// TwinCAT 3 PLC project PLC1
// ProgramVersion: 3.1.4026.16
// libraries:
//   SPT Base Types, * (Beckhoff Automation LLC)
//   Tc2_Standard, * (Beckhoff Automation GmbH)
//   Tc2_System, * (Beckhoff Automation GmbH)
//   Tc3_Module, * (Beckhoff Automation GmbH)
//   Tc3_PackML_V2, * (Beckhoff Automation GmbH)
//   Tc3_XPlanarUtility, * (Beckhoff Automation GmbH)
//   XPlanarApplication, * (Beckhoff Automation LLC)
// project tree:
//   / GlobalTextList.TcGTLO (not stored), PlcTask.TcTTO, Visualization Manager.TcVMO (not stored)
//   POUs/CustomStations/ FB_BounceStation.TcPOU, FB_RotateStation.TcPOU (not stored), FB_TiltStation.TcPOU
//   POUs/ FB_XPlanarModule.TcPOU, MAIN.TcPOU
//   POUs/Utilities/ ErrorStep.TcPOU (not stored), NextMinorStep.TcPOU (not stored), NextStep.TcPOU (not stored)
//   VISUs/ V_Main.TcVIS
// real-time tasks:
//   TASK MC-Task (MET): cycle T#2ms, priority 6, ADS port 355
//   TASK MC-Task (MPT): cycle T#10ms, priority 7, ADS port 356
//   TASK Job Task: cycle default, priority 8
//   TASK PlcTask: cycle T#10ms, priority 20, ADS port 352
//   TASK XPlanar Task_3: cycle T#250us, priority 1, ADS port 350
//   TASK XPlanar Task_4: cycle T#250us, priority 2, ADS port 351
// I/O:
//   DEVICE Device 1 (EtherCAT), AmsNetId 5.85.147.112.2.1
//     Term 1 (EK1200) [EK1200-5000 EtherCAT Power supply (2A E-Bus)]
//       Term 2 (EL9222-9482) [EL9222-9482 Overcurrent protection 24V DC, 2Ch., 8A/2A]
//       Term 3 (EL9222-6600) [EL9222-6600 Overcurrent protection 24V DC, 2Ch., max. 4A, adjustable]
//       Term 4 (EL9011) [EL9011 End Terminal]
//   DEVICE Device 4 (EtherCAT), AmsNetId 5.85.147.112.5.1
//     Term 5 (APS4322-7000) [APS4322-7000 Drive]
//       Term 6 (APS4322-5000) [APS4322-5000 Feedback]
//     Term 7 (APS4322-7000) [APS4322-7000 Drive]
//       Term 8 (APS4322-5000) [APS4322-5000 Feedback]
//     Term 9 (APS4322-7000) [APS4322-7000 Drive]
//       Term 10 (APS4322-5000) [APS4322-5000 Feedback]
//     Term 11 (APS4322-7000) [APS4322-7000 Drive]
//       Term 12 (APS4322-5000) [APS4322-5000 Feedback]
//     Term 13 (APS4322-7000) [APS4322-7000 Drive]
//       Term 14 (APS4322-5000) [APS4322-5000 Feedback]
//     Term 15 (APS4322-7000) [APS4322-7000 Drive]
//       Term 16 (APS4322-5000) [APS4322-5000 Feedback]
// variable links:
//   Device 4 (EtherCAT) <-> TcCOM Objects/XPlanar/Part1/Tile1
//     Term 5 (APS4322-7000)/APS Comm Inputs/CommStatusWord <-> Data Pointer/MoverCommStatusWord
//     Term 5 (APS4322-7000)/APS Comm Inputs/Data {1..4} <-> Data Pointer/MoverCommDataIn[{0..3}]  (4 links)
//     Term 5 (APS4322-7000)/APS Comm Outputs/CommControlWord <-> Data Pointer/MoverCommControlWord
//     Term 5 (APS4322-7000)/APS Comm Outputs/Data 1 <-> Data Pointer/MoverCommDataOut
//     Term 5 (APS4322-7000)/APS Diagdata/DC Link Voltage <-> Data Pointer/DcLinkVoltage
//     Term 5 (APS4322-7000)/APS Diagdata/Power supply current <-> Data Pointer/PowerSupplyCurrent
//     Term 5 (APS4322-7000)/APS Inputs/StatusWord <-> Data Pointer/PowerUnitStatusWord
//     Term 5 (APS4322-7000)/APS Outputs/ControlWord <-> Data Pointer/PowerUnitControlWord
//     Term 5 (APS4322-7000)/APS Outputs/Current D 0X0 <-> Data Pointer/DCurrentSetPoints[0]
//     Term 5 (APS4322-7000)/APS Outputs/Current D 0X1 <-> Data Pointer/DCurrentSetPoints[1]
//     Term 5 (APS4322-7000)/APS Outputs/Current D 0X2 <-> Data Pointer/DCurrentSetPoints[2]
//     Term 5 (APS4322-7000)/APS Outputs/Current D 1X0 <-> Data Pointer/DCurrentSetPoints[6]
//     Term 5 (APS4322-7000)/APS Outputs/Current D 1X1 <-> Data Pointer/DCurrentSetPoints[7]
//     Term 5 (APS4322-7000)/APS Outputs/Current D 1X2 <-> Data Pointer/DCurrentSetPoints[8]
//     Term 5 (APS4322-7000)/APS Outputs/Current D 2X0 <-> Data Pointer/DCurrentSetPoints[12]
//     Term 5 (APS4322-7000)/APS Outputs/Current D 2X1 <-> Data Pointer/DCurrentSetPoints[13]
//     Term 5 (APS4322-7000)/APS Outputs/Current D 2X2 <-> Data Pointer/DCurrentSetPoints[14]
//     Term 5 (APS4322-7000)/APS Outputs/Current D 3X0 <-> Data Pointer/DCurrentSetPoints[18]
//     Term 5 (APS4322-7000)/APS Outputs/Current D 3X1 <-> Data Pointer/DCurrentSetPoints[19]
//     Term 5 (APS4322-7000)/APS Outputs/Current D 3X2 <-> Data Pointer/DCurrentSetPoints[20]
//     Term 5 (APS4322-7000)/APS Outputs/Current D 0Y0 <-> Data Pointer/DCurrentSetPoints[3]
//     Term 5 (APS4322-7000)/APS Outputs/Current D 0Y1 <-> Data Pointer/DCurrentSetPoints[4]
//     Term 5 (APS4322-7000)/APS Outputs/Current D 0Y2 <-> Data Pointer/DCurrentSetPoints[5]
//     Term 5 (APS4322-7000)/APS Outputs/Current D 1Y0 <-> Data Pointer/DCurrentSetPoints[9]
//     Term 5 (APS4322-7000)/APS Outputs/Current D 1Y1 <-> Data Pointer/DCurrentSetPoints[10]
//     Term 5 (APS4322-7000)/APS Outputs/Current D 1Y2 <-> Data Pointer/DCurrentSetPoints[11]
//     Term 5 (APS4322-7000)/APS Outputs/Current D 2Y0 <-> Data Pointer/DCurrentSetPoints[15]
//     Term 5 (APS4322-7000)/APS Outputs/Current D 2Y1 <-> Data Pointer/DCurrentSetPoints[16]
//     Term 5 (APS4322-7000)/APS Outputs/Current D 2Y2 <-> Data Pointer/DCurrentSetPoints[17]
//     Term 5 (APS4322-7000)/APS Outputs/Current D 3Y0 <-> Data Pointer/DCurrentSetPoints[21]
//     Term 5 (APS4322-7000)/APS Outputs/Current D 3Y1 <-> Data Pointer/DCurrentSetPoints[22]
//     Term 5 (APS4322-7000)/APS Outputs/Current D 3Y2 <-> Data Pointer/DCurrentSetPoints[23]
//     Term 5 (APS4322-7000)/APS Outputs/Current Q 0X0 <-> Data Pointer/QCurrentSetPoints[0]
//     Term 5 (APS4322-7000)/APS Outputs/Current Q 0X1 <-> Data Pointer/QCurrentSetPoints[1]
//     Term 5 (APS4322-7000)/APS Outputs/Current Q 0X2 <-> Data Pointer/QCurrentSetPoints[2]
//     Term 5 (APS4322-7000)/APS Outputs/Current Q 1X0 <-> Data Pointer/QCurrentSetPoints[6]
//     Term 5 (APS4322-7000)/APS Outputs/Current Q 1X1 <-> Data Pointer/QCurrentSetPoints[7]
//     Term 5 (APS4322-7000)/APS Outputs/Current Q 1X2 <-> Data Pointer/QCurrentSetPoints[8]
//     Term 5 (APS4322-7000)/APS Outputs/Current Q 2X0 <-> Data Pointer/QCurrentSetPoints[12]
//     Term 5 (APS4322-7000)/APS Outputs/Current Q 2X1 <-> Data Pointer/QCurrentSetPoints[13]
//     Term 5 (APS4322-7000)/APS Outputs/Current Q 2X2 <-> Data Pointer/QCurrentSetPoints[14]
//     Term 5 (APS4322-7000)/APS Outputs/Current Q 3X0 <-> Data Pointer/QCurrentSetPoints[18]
//     Term 5 (APS4322-7000)/APS Outputs/Current Q 3X1 <-> Data Pointer/QCurrentSetPoints[19]
//     Term 5 (APS4322-7000)/APS Outputs/Current Q 3X2 <-> Data Pointer/QCurrentSetPoints[20]
//     Term 5 (APS4322-7000)/APS Outputs/Current Q 0Y0 <-> Data Pointer/QCurrentSetPoints[3]
//     Term 5 (APS4322-7000)/APS Outputs/Current Q 0Y1 <-> Data Pointer/QCurrentSetPoints[4]
//     Term 5 (APS4322-7000)/APS Outputs/Current Q 0Y2 <-> Data Pointer/QCurrentSetPoints[5]
//     Term 5 (APS4322-7000)/APS Outputs/Current Q 1Y0 <-> Data Pointer/QCurrentSetPoints[9]
//     Term 5 (APS4322-7000)/APS Outputs/Current Q 1Y1 <-> Data Pointer/QCurrentSetPoints[10]
//     Term 5 (APS4322-7000)/APS Outputs/Current Q 1Y2 <-> Data Pointer/QCurrentSetPoints[11]
//     Term 5 (APS4322-7000)/APS Outputs/Current Q 2Y0 <-> Data Pointer/QCurrentSetPoints[15]
//     Term 5 (APS4322-7000)/APS Outputs/Current Q 2Y1 <-> Data Pointer/QCurrentSetPoints[16]
//     Term 5 (APS4322-7000)/APS Outputs/Current Q 2Y2 <-> Data Pointer/QCurrentSetPoints[17]
//     Term 5 (APS4322-7000)/APS Outputs/Current Q 3Y0 <-> Data Pointer/QCurrentSetPoints[21]
//     Term 5 (APS4322-7000)/APS Outputs/Current Q 3Y1 <-> Data Pointer/QCurrentSetPoints[22]
//     Term 5 (APS4322-7000)/APS Outputs/Current Q 3Y2 <-> Data Pointer/QCurrentSetPoints[23]
//     Term 5 (APS4322-7000)/APS Outputs/PhiE 0X0 <-> Data Pointer/PhiSetPoints[0]
//     Term 5 (APS4322-7000)/APS Outputs/PhiE 0X1 <-> Data Pointer/PhiSetPoints[1]
//     Term 5 (APS4322-7000)/APS Outputs/PhiE 0X2 <-> Data Pointer/PhiSetPoints[2]
//     Term 5 (APS4322-7000)/APS Outputs/PhiE 1X0 <-> Data Pointer/PhiSetPoints[6]
//     Term 5 (APS4322-7000)/APS Outputs/PhiE 1X1 <-> Data Pointer/PhiSetPoints[7]
//     Term 5 (APS4322-7000)/APS Outputs/PhiE 1X2 <-> Data Pointer/PhiSetPoints[8]
//     Term 5 (APS4322-7000)/APS Outputs/PhiE 2X0 <-> Data Pointer/PhiSetPoints[12]
//     Term 5 (APS4322-7000)/APS Outputs/PhiE 2X1 <-> Data Pointer/PhiSetPoints[13]
//     Term 5 (APS4322-7000)/APS Outputs/PhiE 2X2 <-> Data Pointer/PhiSetPoints[14]
//     Term 5 (APS4322-7000)/APS Outputs/PhiE 3X0 <-> Data Pointer/PhiSetPoints[18]
//     Term 5 (APS4322-7000)/APS Outputs/PhiE 3X1 <-> Data Pointer/PhiSetPoints[19]
//     Term 5 (APS4322-7000)/APS Outputs/PhiE 3X2 <-> Data Pointer/PhiSetPoints[20]
//     Term 5 (APS4322-7000)/APS Outputs/PhiE 0Y0 <-> Data Pointer/PhiSetPoints[3]
//     Term 5 (APS4322-7000)/APS Outputs/PhiE 0Y1 <-> Data Pointer/PhiSetPoints[4]
//     Term 5 (APS4322-7000)/APS Outputs/PhiE 0Y2 <-> Data Pointer/PhiSetPoints[5]
//     Term 5 (APS4322-7000)/APS Outputs/PhiE 1Y0 <-> Data Pointer/PhiSetPoints[9]
//     Term 5 (APS4322-7000)/APS Outputs/PhiE 1Y1 <-> Data Pointer/PhiSetPoints[10]
//     Term 5 (APS4322-7000)/APS Outputs/PhiE 1Y2 <-> Data Pointer/PhiSetPoints[11]
//     Term 5 (APS4322-7000)/APS Outputs/PhiE 2Y0 <-> Data Pointer/PhiSetPoints[15]
//     Term 5 (APS4322-7000)/APS Outputs/PhiE 2Y1 <-> Data Pointer/PhiSetPoints[16]
//     Term 5 (APS4322-7000)/APS Outputs/PhiE 2Y2 <-> Data Pointer/PhiSetPoints[17]
//     Term 5 (APS4322-7000)/APS Outputs/PhiE 3Y0 <-> Data Pointer/PhiSetPoints[21]
//     Term 5 (APS4322-7000)/APS Outputs/PhiE 3Y1 <-> Data Pointer/PhiSetPoints[22]
//     Term 5 (APS4322-7000)/APS Outputs/PhiE 3Y2 <-> Data Pointer/PhiSetPoints[23]
//     Term 5 (APS4322-7000)/Term 6 (APS4322-5000)/FB Inputs/A{0..8 step 2} X-Field <-> Data Pointer/HallSensorFieldsXYZ[{0..12 step 3}]  (5 links)
//     Term 5 (APS4322-7000)/Term 6 (APS4322-5000)/FB Inputs/A{0..8 step 2} Y-Field <-> Data Pointer/HallSensorFieldsXYZ[{1..13 step 3}]  (5 links)
//     Term 5 (APS4322-7000)/Term 6 (APS4322-5000)/FB Inputs/A{0..8 step 2} Z-Field <-> Data Pointer/HallSensorFieldsXYZ[{2..14 step 3}]  (5 links)
//     Term 5 (APS4322-7000)/Term 6 (APS4322-5000)/FB Inputs/B{1..9 step 2} X-Field <-> Data Pointer/HallSensorFieldsXYZ[{15..27 step 3}]  (5 links)
//     Term 5 (APS4322-7000)/Term 6 (APS4322-5000)/FB Inputs/B{1..9 step 2} Y-Field <-> Data Pointer/HallSensorFieldsXYZ[{16..28 step 3}]  (5 links)
//     Term 5 (APS4322-7000)/Term 6 (APS4322-5000)/FB Inputs/B{1..9 step 2} Z-Field <-> Data Pointer/HallSensorFieldsXYZ[{17..29 step 3}]  (5 links)
//     Term 5 (APS4322-7000)/Term 6 (APS4322-5000)/FB Inputs/C{0..8 step 2} X-Field <-> Data Pointer/HallSensorFieldsXYZ[{30..42 step 3}]  (5 links)
//     Term 5 (APS4322-7000)/Term 6 (APS4322-5000)/FB Inputs/C{0..8 step 2} Y-Field <-> Data Pointer/HallSensorFieldsXYZ[{31..43 step 3}]  (5 links)
//     Term 5 (APS4322-7000)/Term 6 (APS4322-5000)/FB Inputs/C{0..8 step 2} Z-Field <-> Data Pointer/HallSensorFieldsXYZ[{32..44 step 3}]  (5 links)
//     Term 5 (APS4322-7000)/Term 6 (APS4322-5000)/FB Inputs/D{1..9 step 2} X-Field <-> Data Pointer/HallSensorFieldsXYZ[{45..57 step 3}]  (5 links)
//     Term 5 (APS4322-7000)/Term 6 (APS4322-5000)/FB Inputs/D{1..9 step 2} Y-Field <-> Data Pointer/HallSensorFieldsXYZ[{46..58 step 3}]  (5 links)
//     Term 5 (APS4322-7000)/Term 6 (APS4322-5000)/FB Inputs/D{1..9 step 2} Z-Field <-> Data Pointer/HallSensorFieldsXYZ[{47..59 step 3}]  (5 links)
//     Term 5 (APS4322-7000)/Term 6 (APS4322-5000)/FB Inputs/E{0..8 step 2} X-Field <-> Data Pointer/HallSensorFieldsXYZ[{60..72 step 3}]  (5 links)
//     Term 5 (APS4322-7000)/Term 6 (APS4322-5000)/FB Inputs/E{0..8 step 2} Y-Field <-> Data Pointer/HallSensorFieldsXYZ[{61..73 step 3}]  (5 links)
//     Term 5 (APS4322-7000)/Term 6 (APS4322-5000)/FB Inputs/E{0..8 step 2} Z-Field <-> Data Pointer/HallSensorFieldsXYZ[{62..74 step 3}]  (5 links)
//     Term 5 (APS4322-7000)/Term 6 (APS4322-5000)/FB Inputs/F{1..9 step 2} X-Field <-> Data Pointer/HallSensorFieldsXYZ[{75..87 step 3}]  (5 links)
//     Term 5 (APS4322-7000)/Term 6 (APS4322-5000)/FB Inputs/F{1..9 step 2} Y-Field <-> Data Pointer/HallSensorFieldsXYZ[{76..88 step 3}]  (5 links)
//     Term 5 (APS4322-7000)/Term 6 (APS4322-5000)/FB Inputs/F{1..9 step 2} Z-Field <-> Data Pointer/HallSensorFieldsXYZ[{77..89 step 3}]  (5 links)
//     Term 5 (APS4322-7000)/Term 6 (APS4322-5000)/FB Inputs/G{0..8 step 2} X-Field <-> Data Pointer/HallSensorFieldsXYZ[{90..102 step 3}]  (5 links)
//     Term 5 (APS4322-7000)/Term 6 (APS4322-5000)/FB Inputs/G{0..8 step 2} Y-Field <-> Data Pointer/HallSensorFieldsXYZ[{91..103 step 3}]  (5 links)
//     Term 5 (APS4322-7000)/Term 6 (APS4322-5000)/FB Inputs/G{0..8 step 2} Z-Field <-> Data Pointer/HallSensorFieldsXYZ[{92..104 step 3}]  (5 links)
//     Term 5 (APS4322-7000)/Term 6 (APS4322-5000)/FB Inputs/H{1..9 step 2} X-Field <-> Data Pointer/HallSensorFieldsXYZ[{105..117 step 3}]  (5 links)
//     Term 5 (APS4322-7000)/Term 6 (APS4322-5000)/FB Inputs/H{1..9 step 2} Y-Field <-> Data Pointer/HallSensorFieldsXYZ[{106..118 step 3}]  (5 links)
//     Term 5 (APS4322-7000)/Term 6 (APS4322-5000)/FB Inputs/H{1..9 step 2} Z-Field <-> Data Pointer/HallSensorFieldsXYZ[{107..119 step 3}]  (5 links)
//     Term 5 (APS4322-7000)/Term 6 (APS4322-5000)/FB Inputs/I{0..8 step 2} X-Field <-> Data Pointer/HallSensorFieldsXYZ[{120..132 step 3}]  (5 links)
//     Term 5 (APS4322-7000)/Term 6 (APS4322-5000)/FB Inputs/I{0..8 step 2} Y-Field <-> Data Pointer/HallSensorFieldsXYZ[{121..133 step 3}]  (5 links)
//     Term 5 (APS4322-7000)/Term 6 (APS4322-5000)/FB Inputs/I{0..8 step 2} Z-Field <-> Data Pointer/HallSensorFieldsXYZ[{122..134 step 3}]  (5 links)
//     Term 5 (APS4322-7000)/Term 6 (APS4322-5000)/FB Inputs/J{1..9 step 2} X-Field <-> Data Pointer/HallSensorFieldsXYZ[{135..147 step 3}]  (5 links)
//     Term 5 (APS4322-7000)/Term 6 (APS4322-5000)/FB Inputs/J{1..9 step 2} Y-Field <-> Data Pointer/HallSensorFieldsXYZ[{136..148 step 3}]  (5 links)
//     Term 5 (APS4322-7000)/Term 6 (APS4322-5000)/FB Inputs/J{1..9 step 2} Z-Field <-> Data Pointer/HallSensorFieldsXYZ[{137..149 step 3}]  (5 links)
//     Term 5 (APS4322-7000)/Term 6 (APS4322-5000)/FB Inputs/Status <-> Data Pointer/FeedbackStatus
//   Device 4 (EtherCAT) <-> TcCOM Objects/XPlanar/Part1/Tile2
//     Term 7 (APS4322-7000)/APS Comm Inputs/CommStatusWord <-> Data Pointer/MoverCommStatusWord
//     Term 7 (APS4322-7000)/APS Comm Inputs/Data {1..4} <-> Data Pointer/MoverCommDataIn[{0..3}]  (4 links)
//     Term 7 (APS4322-7000)/APS Comm Outputs/CommControlWord <-> Data Pointer/MoverCommControlWord
//     Term 7 (APS4322-7000)/APS Comm Outputs/Data 1 <-> Data Pointer/MoverCommDataOut
//     Term 7 (APS4322-7000)/APS Diagdata/DC Link Voltage <-> Data Pointer/DcLinkVoltage
//     Term 7 (APS4322-7000)/APS Diagdata/Power supply current <-> Data Pointer/PowerSupplyCurrent
//     Term 7 (APS4322-7000)/APS Inputs/StatusWord <-> Data Pointer/PowerUnitStatusWord
//     Term 7 (APS4322-7000)/APS Outputs/ControlWord <-> Data Pointer/PowerUnitControlWord
//     Term 7 (APS4322-7000)/APS Outputs/Current D 0X0 <-> Data Pointer/DCurrentSetPoints[0]
//     Term 7 (APS4322-7000)/APS Outputs/Current D 0X1 <-> Data Pointer/DCurrentSetPoints[1]
//     Term 7 (APS4322-7000)/APS Outputs/Current D 0X2 <-> Data Pointer/DCurrentSetPoints[2]
//     Term 7 (APS4322-7000)/APS Outputs/Current D 1X0 <-> Data Pointer/DCurrentSetPoints[6]
//     Term 7 (APS4322-7000)/APS Outputs/Current D 1X1 <-> Data Pointer/DCurrentSetPoints[7]
//     Term 7 (APS4322-7000)/APS Outputs/Current D 1X2 <-> Data Pointer/DCurrentSetPoints[8]
//     Term 7 (APS4322-7000)/APS Outputs/Current D 2X0 <-> Data Pointer/DCurrentSetPoints[12]
//     Term 7 (APS4322-7000)/APS Outputs/Current D 2X1 <-> Data Pointer/DCurrentSetPoints[13]
//     Term 7 (APS4322-7000)/APS Outputs/Current D 2X2 <-> Data Pointer/DCurrentSetPoints[14]
//     Term 7 (APS4322-7000)/APS Outputs/Current D 3X0 <-> Data Pointer/DCurrentSetPoints[18]
//     Term 7 (APS4322-7000)/APS Outputs/Current D 3X1 <-> Data Pointer/DCurrentSetPoints[19]
//     Term 7 (APS4322-7000)/APS Outputs/Current D 3X2 <-> Data Pointer/DCurrentSetPoints[20]
//     Term 7 (APS4322-7000)/APS Outputs/Current D 0Y0 <-> Data Pointer/DCurrentSetPoints[3]
//     Term 7 (APS4322-7000)/APS Outputs/Current D 0Y1 <-> Data Pointer/DCurrentSetPoints[4]
//     Term 7 (APS4322-7000)/APS Outputs/Current D 0Y2 <-> Data Pointer/DCurrentSetPoints[5]
//     Term 7 (APS4322-7000)/APS Outputs/Current D 1Y0 <-> Data Pointer/DCurrentSetPoints[9]
//     Term 7 (APS4322-7000)/APS Outputs/Current D 1Y1 <-> Data Pointer/DCurrentSetPoints[10]
//     Term 7 (APS4322-7000)/APS Outputs/Current D 1Y2 <-> Data Pointer/DCurrentSetPoints[11]
//     Term 7 (APS4322-7000)/APS Outputs/Current D 2Y0 <-> Data Pointer/DCurrentSetPoints[15]
//     Term 7 (APS4322-7000)/APS Outputs/Current D 2Y1 <-> Data Pointer/DCurrentSetPoints[16]
//     Term 7 (APS4322-7000)/APS Outputs/Current D 2Y2 <-> Data Pointer/DCurrentSetPoints[17]
//     Term 7 (APS4322-7000)/APS Outputs/Current D 3Y0 <-> Data Pointer/DCurrentSetPoints[21]
//     Term 7 (APS4322-7000)/APS Outputs/Current D 3Y1 <-> Data Pointer/DCurrentSetPoints[22]
//     Term 7 (APS4322-7000)/APS Outputs/Current D 3Y2 <-> Data Pointer/DCurrentSetPoints[23]
//     Term 7 (APS4322-7000)/APS Outputs/Current Q 0X0 <-> Data Pointer/QCurrentSetPoints[0]
//     Term 7 (APS4322-7000)/APS Outputs/Current Q 0X1 <-> Data Pointer/QCurrentSetPoints[1]
//     Term 7 (APS4322-7000)/APS Outputs/Current Q 0X2 <-> Data Pointer/QCurrentSetPoints[2]
//     Term 7 (APS4322-7000)/APS Outputs/Current Q 1X0 <-> Data Pointer/QCurrentSetPoints[6]
//     Term 7 (APS4322-7000)/APS Outputs/Current Q 1X1 <-> Data Pointer/QCurrentSetPoints[7]
//     Term 7 (APS4322-7000)/APS Outputs/Current Q 1X2 <-> Data Pointer/QCurrentSetPoints[8]
//     Term 7 (APS4322-7000)/APS Outputs/Current Q 2X0 <-> Data Pointer/QCurrentSetPoints[12]
//     Term 7 (APS4322-7000)/APS Outputs/Current Q 2X1 <-> Data Pointer/QCurrentSetPoints[13]
//     Term 7 (APS4322-7000)/APS Outputs/Current Q 2X2 <-> Data Pointer/QCurrentSetPoints[14]
//     Term 7 (APS4322-7000)/APS Outputs/Current Q 3X0 <-> Data Pointer/QCurrentSetPoints[18]
//     Term 7 (APS4322-7000)/APS Outputs/Current Q 3X1 <-> Data Pointer/QCurrentSetPoints[19]
//     Term 7 (APS4322-7000)/APS Outputs/Current Q 3X2 <-> Data Pointer/QCurrentSetPoints[20]
//     Term 7 (APS4322-7000)/APS Outputs/Current Q 0Y0 <-> Data Pointer/QCurrentSetPoints[3]
//     Term 7 (APS4322-7000)/APS Outputs/Current Q 0Y1 <-> Data Pointer/QCurrentSetPoints[4]
//     Term 7 (APS4322-7000)/APS Outputs/Current Q 0Y2 <-> Data Pointer/QCurrentSetPoints[5]
//     Term 7 (APS4322-7000)/APS Outputs/Current Q 1Y0 <-> Data Pointer/QCurrentSetPoints[9]
//     Term 7 (APS4322-7000)/APS Outputs/Current Q 1Y1 <-> Data Pointer/QCurrentSetPoints[10]
//     Term 7 (APS4322-7000)/APS Outputs/Current Q 1Y2 <-> Data Pointer/QCurrentSetPoints[11]
//     Term 7 (APS4322-7000)/APS Outputs/Current Q 2Y0 <-> Data Pointer/QCurrentSetPoints[15]
//     Term 7 (APS4322-7000)/APS Outputs/Current Q 2Y1 <-> Data Pointer/QCurrentSetPoints[16]
//     Term 7 (APS4322-7000)/APS Outputs/Current Q 2Y2 <-> Data Pointer/QCurrentSetPoints[17]
//     Term 7 (APS4322-7000)/APS Outputs/Current Q 3Y0 <-> Data Pointer/QCurrentSetPoints[21]
//     Term 7 (APS4322-7000)/APS Outputs/Current Q 3Y1 <-> Data Pointer/QCurrentSetPoints[22]
//     Term 7 (APS4322-7000)/APS Outputs/Current Q 3Y2 <-> Data Pointer/QCurrentSetPoints[23]
//     Term 7 (APS4322-7000)/APS Outputs/PhiE 0X0 <-> Data Pointer/PhiSetPoints[0]
//     Term 7 (APS4322-7000)/APS Outputs/PhiE 0X1 <-> Data Pointer/PhiSetPoints[1]
//     Term 7 (APS4322-7000)/APS Outputs/PhiE 0X2 <-> Data Pointer/PhiSetPoints[2]
//     Term 7 (APS4322-7000)/APS Outputs/PhiE 1X0 <-> Data Pointer/PhiSetPoints[6]
//     Term 7 (APS4322-7000)/APS Outputs/PhiE 1X1 <-> Data Pointer/PhiSetPoints[7]
//     Term 7 (APS4322-7000)/APS Outputs/PhiE 1X2 <-> Data Pointer/PhiSetPoints[8]
//     Term 7 (APS4322-7000)/APS Outputs/PhiE 2X0 <-> Data Pointer/PhiSetPoints[12]
//     Term 7 (APS4322-7000)/APS Outputs/PhiE 2X1 <-> Data Pointer/PhiSetPoints[13]
//     Term 7 (APS4322-7000)/APS Outputs/PhiE 2X2 <-> Data Pointer/PhiSetPoints[14]
//     Term 7 (APS4322-7000)/APS Outputs/PhiE 3X0 <-> Data Pointer/PhiSetPoints[18]
//     Term 7 (APS4322-7000)/APS Outputs/PhiE 3X1 <-> Data Pointer/PhiSetPoints[19]
//     Term 7 (APS4322-7000)/APS Outputs/PhiE 3X2 <-> Data Pointer/PhiSetPoints[20]
//     Term 7 (APS4322-7000)/APS Outputs/PhiE 0Y0 <-> Data Pointer/PhiSetPoints[3]
//     Term 7 (APS4322-7000)/APS Outputs/PhiE 0Y1 <-> Data Pointer/PhiSetPoints[4]
//     Term 7 (APS4322-7000)/APS Outputs/PhiE 0Y2 <-> Data Pointer/PhiSetPoints[5]
//     Term 7 (APS4322-7000)/APS Outputs/PhiE 1Y0 <-> Data Pointer/PhiSetPoints[9]
//     Term 7 (APS4322-7000)/APS Outputs/PhiE 1Y1 <-> Data Pointer/PhiSetPoints[10]
//     Term 7 (APS4322-7000)/APS Outputs/PhiE 1Y2 <-> Data Pointer/PhiSetPoints[11]
//     Term 7 (APS4322-7000)/APS Outputs/PhiE 2Y0 <-> Data Pointer/PhiSetPoints[15]
//     Term 7 (APS4322-7000)/APS Outputs/PhiE 2Y1 <-> Data Pointer/PhiSetPoints[16]
//     Term 7 (APS4322-7000)/APS Outputs/PhiE 2Y2 <-> Data Pointer/PhiSetPoints[17]
//     Term 7 (APS4322-7000)/APS Outputs/PhiE 3Y0 <-> Data Pointer/PhiSetPoints[21]
//     Term 7 (APS4322-7000)/APS Outputs/PhiE 3Y1 <-> Data Pointer/PhiSetPoints[22]
//     Term 7 (APS4322-7000)/APS Outputs/PhiE 3Y2 <-> Data Pointer/PhiSetPoints[23]
//     Term 7 (APS4322-7000)/Term 8 (APS4322-5000)/FB Inputs/A{0..8 step 2} X-Field <-> Data Pointer/HallSensorFieldsXYZ[{0..12 step 3}]  (5 links)
//     Term 7 (APS4322-7000)/Term 8 (APS4322-5000)/FB Inputs/A{0..8 step 2} Y-Field <-> Data Pointer/HallSensorFieldsXYZ[{1..13 step 3}]  (5 links)
//     Term 7 (APS4322-7000)/Term 8 (APS4322-5000)/FB Inputs/A{0..8 step 2} Z-Field <-> Data Pointer/HallSensorFieldsXYZ[{2..14 step 3}]  (5 links)
//     Term 7 (APS4322-7000)/Term 8 (APS4322-5000)/FB Inputs/B{1..9 step 2} X-Field <-> Data Pointer/HallSensorFieldsXYZ[{15..27 step 3}]  (5 links)
//     Term 7 (APS4322-7000)/Term 8 (APS4322-5000)/FB Inputs/B{1..9 step 2} Y-Field <-> Data Pointer/HallSensorFieldsXYZ[{16..28 step 3}]  (5 links)
//     Term 7 (APS4322-7000)/Term 8 (APS4322-5000)/FB Inputs/B{1..9 step 2} Z-Field <-> Data Pointer/HallSensorFieldsXYZ[{17..29 step 3}]  (5 links)
//     Term 7 (APS4322-7000)/Term 8 (APS4322-5000)/FB Inputs/C{0..8 step 2} X-Field <-> Data Pointer/HallSensorFieldsXYZ[{30..42 step 3}]  (5 links)
//     Term 7 (APS4322-7000)/Term 8 (APS4322-5000)/FB Inputs/C{0..8 step 2} Y-Field <-> Data Pointer/HallSensorFieldsXYZ[{31..43 step 3}]  (5 links)
//     Term 7 (APS4322-7000)/Term 8 (APS4322-5000)/FB Inputs/C{0..8 step 2} Z-Field <-> Data Pointer/HallSensorFieldsXYZ[{32..44 step 3}]  (5 links)
//     Term 7 (APS4322-7000)/Term 8 (APS4322-5000)/FB Inputs/D{1..9 step 2} X-Field <-> Data Pointer/HallSensorFieldsXYZ[{45..57 step 3}]  (5 links)
//     Term 7 (APS4322-7000)/Term 8 (APS4322-5000)/FB Inputs/D{1..9 step 2} Y-Field <-> Data Pointer/HallSensorFieldsXYZ[{46..58 step 3}]  (5 links)
//     Term 7 (APS4322-7000)/Term 8 (APS4322-5000)/FB Inputs/D{1..9 step 2} Z-Field <-> Data Pointer/HallSensorFieldsXYZ[{47..59 step 3}]  (5 links)
//     Term 7 (APS4322-7000)/Term 8 (APS4322-5000)/FB Inputs/E{0..8 step 2} X-Field <-> Data Pointer/HallSensorFieldsXYZ[{60..72 step 3}]  (5 links)
//     Term 7 (APS4322-7000)/Term 8 (APS4322-5000)/FB Inputs/E{0..8 step 2} Y-Field <-> Data Pointer/HallSensorFieldsXYZ[{61..73 step 3}]  (5 links)
//     Term 7 (APS4322-7000)/Term 8 (APS4322-5000)/FB Inputs/E{0..8 step 2} Z-Field <-> Data Pointer/HallSensorFieldsXYZ[{62..74 step 3}]  (5 links)
//     Term 7 (APS4322-7000)/Term 8 (APS4322-5000)/FB Inputs/F{1..9 step 2} X-Field <-> Data Pointer/HallSensorFieldsXYZ[{75..87 step 3}]  (5 links)
//     Term 7 (APS4322-7000)/Term 8 (APS4322-5000)/FB Inputs/F{1..9 step 2} Y-Field <-> Data Pointer/HallSensorFieldsXYZ[{76..88 step 3}]  (5 links)
//     Term 7 (APS4322-7000)/Term 8 (APS4322-5000)/FB Inputs/F{1..9 step 2} Z-Field <-> Data Pointer/HallSensorFieldsXYZ[{77..89 step 3}]  (5 links)
//     Term 7 (APS4322-7000)/Term 8 (APS4322-5000)/FB Inputs/G{0..8 step 2} X-Field <-> Data Pointer/HallSensorFieldsXYZ[{90..102 step 3}]  (5 links)
//     Term 7 (APS4322-7000)/Term 8 (APS4322-5000)/FB Inputs/G{0..8 step 2} Y-Field <-> Data Pointer/HallSensorFieldsXYZ[{91..103 step 3}]  (5 links)
//     Term 7 (APS4322-7000)/Term 8 (APS4322-5000)/FB Inputs/G{0..8 step 2} Z-Field <-> Data Pointer/HallSensorFieldsXYZ[{92..104 step 3}]  (5 links)
//     Term 7 (APS4322-7000)/Term 8 (APS4322-5000)/FB Inputs/H{1..9 step 2} X-Field <-> Data Pointer/HallSensorFieldsXYZ[{105..117 step 3}]  (5 links)
//     Term 7 (APS4322-7000)/Term 8 (APS4322-5000)/FB Inputs/H{1..9 step 2} Y-Field <-> Data Pointer/HallSensorFieldsXYZ[{106..118 step 3}]  (5 links)
//     Term 7 (APS4322-7000)/Term 8 (APS4322-5000)/FB Inputs/H{1..9 step 2} Z-Field <-> Data Pointer/HallSensorFieldsXYZ[{107..119 step 3}]  (5 links)
//     Term 7 (APS4322-7000)/Term 8 (APS4322-5000)/FB Inputs/I{0..8 step 2} X-Field <-> Data Pointer/HallSensorFieldsXYZ[{120..132 step 3}]  (5 links)
//     Term 7 (APS4322-7000)/Term 8 (APS4322-5000)/FB Inputs/I{0..8 step 2} Y-Field <-> Data Pointer/HallSensorFieldsXYZ[{121..133 step 3}]  (5 links)
//     Term 7 (APS4322-7000)/Term 8 (APS4322-5000)/FB Inputs/I{0..8 step 2} Z-Field <-> Data Pointer/HallSensorFieldsXYZ[{122..134 step 3}]  (5 links)
//     Term 7 (APS4322-7000)/Term 8 (APS4322-5000)/FB Inputs/J{1..9 step 2} X-Field <-> Data Pointer/HallSensorFieldsXYZ[{135..147 step 3}]  (5 links)
//     Term 7 (APS4322-7000)/Term 8 (APS4322-5000)/FB Inputs/J{1..9 step 2} Y-Field <-> Data Pointer/HallSensorFieldsXYZ[{136..148 step 3}]  (5 links)
//     Term 7 (APS4322-7000)/Term 8 (APS4322-5000)/FB Inputs/J{1..9 step 2} Z-Field <-> Data Pointer/HallSensorFieldsXYZ[{137..149 step 3}]  (5 links)
//     Term 7 (APS4322-7000)/Term 8 (APS4322-5000)/FB Inputs/Status <-> Data Pointer/FeedbackStatus
//   Device 4 (EtherCAT) <-> TcCOM Objects/XPlanar/Part1/Tile3
//     Term 9 (APS4322-7000)/APS Comm Inputs/CommStatusWord <-> Data Pointer/MoverCommStatusWord
//     Term 9 (APS4322-7000)/APS Comm Inputs/Data {1..4} <-> Data Pointer/MoverCommDataIn[{0..3}]  (4 links)
//     Term 9 (APS4322-7000)/APS Comm Outputs/CommControlWord <-> Data Pointer/MoverCommControlWord
//     Term 9 (APS4322-7000)/APS Comm Outputs/Data 1 <-> Data Pointer/MoverCommDataOut
//     Term 9 (APS4322-7000)/APS Diagdata/DC Link Voltage <-> Data Pointer/DcLinkVoltage
//     Term 9 (APS4322-7000)/APS Diagdata/Power supply current <-> Data Pointer/PowerSupplyCurrent
//     Term 9 (APS4322-7000)/APS Inputs/StatusWord <-> Data Pointer/PowerUnitStatusWord
//     Term 9 (APS4322-7000)/APS Outputs/ControlWord <-> Data Pointer/PowerUnitControlWord
//     Term 9 (APS4322-7000)/APS Outputs/Current D 0X0 <-> Data Pointer/DCurrentSetPoints[0]
//     Term 9 (APS4322-7000)/APS Outputs/Current D 0X1 <-> Data Pointer/DCurrentSetPoints[1]
//     Term 9 (APS4322-7000)/APS Outputs/Current D 0X2 <-> Data Pointer/DCurrentSetPoints[2]
//     Term 9 (APS4322-7000)/APS Outputs/Current D 1X0 <-> Data Pointer/DCurrentSetPoints[6]
//     Term 9 (APS4322-7000)/APS Outputs/Current D 1X1 <-> Data Pointer/DCurrentSetPoints[7]
//     Term 9 (APS4322-7000)/APS Outputs/Current D 1X2 <-> Data Pointer/DCurrentSetPoints[8]
//     Term 9 (APS4322-7000)/APS Outputs/Current D 2X0 <-> Data Pointer/DCurrentSetPoints[12]
//     Term 9 (APS4322-7000)/APS Outputs/Current D 2X1 <-> Data Pointer/DCurrentSetPoints[13]
//     Term 9 (APS4322-7000)/APS Outputs/Current D 2X2 <-> Data Pointer/DCurrentSetPoints[14]
//     Term 9 (APS4322-7000)/APS Outputs/Current D 3X0 <-> Data Pointer/DCurrentSetPoints[18]
//     Term 9 (APS4322-7000)/APS Outputs/Current D 3X1 <-> Data Pointer/DCurrentSetPoints[19]
//     Term 9 (APS4322-7000)/APS Outputs/Current D 3X2 <-> Data Pointer/DCurrentSetPoints[20]
//     Term 9 (APS4322-7000)/APS Outputs/Current D 0Y0 <-> Data Pointer/DCurrentSetPoints[3]
//     Term 9 (APS4322-7000)/APS Outputs/Current D 0Y1 <-> Data Pointer/DCurrentSetPoints[4]
//     Term 9 (APS4322-7000)/APS Outputs/Current D 0Y2 <-> Data Pointer/DCurrentSetPoints[5]
//     Term 9 (APS4322-7000)/APS Outputs/Current D 1Y0 <-> Data Pointer/DCurrentSetPoints[9]
//     Term 9 (APS4322-7000)/APS Outputs/Current D 1Y1 <-> Data Pointer/DCurrentSetPoints[10]
//     Term 9 (APS4322-7000)/APS Outputs/Current D 1Y2 <-> Data Pointer/DCurrentSetPoints[11]
//     Term 9 (APS4322-7000)/APS Outputs/Current D 2Y0 <-> Data Pointer/DCurrentSetPoints[15]
//     Term 9 (APS4322-7000)/APS Outputs/Current D 2Y1 <-> Data Pointer/DCurrentSetPoints[16]
//     Term 9 (APS4322-7000)/APS Outputs/Current D 2Y2 <-> Data Pointer/DCurrentSetPoints[17]
//     Term 9 (APS4322-7000)/APS Outputs/Current D 3Y0 <-> Data Pointer/DCurrentSetPoints[21]
//     Term 9 (APS4322-7000)/APS Outputs/Current D 3Y1 <-> Data Pointer/DCurrentSetPoints[22]
//     Term 9 (APS4322-7000)/APS Outputs/Current D 3Y2 <-> Data Pointer/DCurrentSetPoints[23]
//     Term 9 (APS4322-7000)/APS Outputs/Current Q 0X0 <-> Data Pointer/QCurrentSetPoints[0]
//     Term 9 (APS4322-7000)/APS Outputs/Current Q 0X1 <-> Data Pointer/QCurrentSetPoints[1]
//     Term 9 (APS4322-7000)/APS Outputs/Current Q 0X2 <-> Data Pointer/QCurrentSetPoints[2]
//     Term 9 (APS4322-7000)/APS Outputs/Current Q 1X0 <-> Data Pointer/QCurrentSetPoints[6]
//     Term 9 (APS4322-7000)/APS Outputs/Current Q 1X1 <-> Data Pointer/QCurrentSetPoints[7]
//     Term 9 (APS4322-7000)/APS Outputs/Current Q 1X2 <-> Data Pointer/QCurrentSetPoints[8]
//     Term 9 (APS4322-7000)/APS Outputs/Current Q 2X0 <-> Data Pointer/QCurrentSetPoints[12]
//     Term 9 (APS4322-7000)/APS Outputs/Current Q 2X1 <-> Data Pointer/QCurrentSetPoints[13]
//     Term 9 (APS4322-7000)/APS Outputs/Current Q 2X2 <-> Data Pointer/QCurrentSetPoints[14]
//     Term 9 (APS4322-7000)/APS Outputs/Current Q 3X0 <-> Data Pointer/QCurrentSetPoints[18]
//     Term 9 (APS4322-7000)/APS Outputs/Current Q 3X1 <-> Data Pointer/QCurrentSetPoints[19]
//     Term 9 (APS4322-7000)/APS Outputs/Current Q 3X2 <-> Data Pointer/QCurrentSetPoints[20]
//     Term 9 (APS4322-7000)/APS Outputs/Current Q 0Y0 <-> Data Pointer/QCurrentSetPoints[3]
//     Term 9 (APS4322-7000)/APS Outputs/Current Q 0Y1 <-> Data Pointer/QCurrentSetPoints[4]
//     Term 9 (APS4322-7000)/APS Outputs/Current Q 0Y2 <-> Data Pointer/QCurrentSetPoints[5]
//     Term 9 (APS4322-7000)/APS Outputs/Current Q 1Y0 <-> Data Pointer/QCurrentSetPoints[9]
//     Term 9 (APS4322-7000)/APS Outputs/Current Q 1Y1 <-> Data Pointer/QCurrentSetPoints[10]
//     Term 9 (APS4322-7000)/APS Outputs/Current Q 1Y2 <-> Data Pointer/QCurrentSetPoints[11]
//     Term 9 (APS4322-7000)/APS Outputs/Current Q 2Y0 <-> Data Pointer/QCurrentSetPoints[15]
//     Term 9 (APS4322-7000)/APS Outputs/Current Q 2Y1 <-> Data Pointer/QCurrentSetPoints[16]
//     Term 9 (APS4322-7000)/APS Outputs/Current Q 2Y2 <-> Data Pointer/QCurrentSetPoints[17]
//     Term 9 (APS4322-7000)/APS Outputs/Current Q 3Y0 <-> Data Pointer/QCurrentSetPoints[21]
//     Term 9 (APS4322-7000)/APS Outputs/Current Q 3Y1 <-> Data Pointer/QCurrentSetPoints[22]
//     Term 9 (APS4322-7000)/APS Outputs/Current Q 3Y2 <-> Data Pointer/QCurrentSetPoints[23]
//     Term 9 (APS4322-7000)/APS Outputs/PhiE 0X0 <-> Data Pointer/PhiSetPoints[0]
//     Term 9 (APS4322-7000)/APS Outputs/PhiE 0X1 <-> Data Pointer/PhiSetPoints[1]
//     Term 9 (APS4322-7000)/APS Outputs/PhiE 0X2 <-> Data Pointer/PhiSetPoints[2]
//     Term 9 (APS4322-7000)/APS Outputs/PhiE 1X0 <-> Data Pointer/PhiSetPoints[6]
//     Term 9 (APS4322-7000)/APS Outputs/PhiE 1X1 <-> Data Pointer/PhiSetPoints[7]
//     Term 9 (APS4322-7000)/APS Outputs/PhiE 1X2 <-> Data Pointer/PhiSetPoints[8]
//     Term 9 (APS4322-7000)/APS Outputs/PhiE 2X0 <-> Data Pointer/PhiSetPoints[12]
//     Term 9 (APS4322-7000)/APS Outputs/PhiE 2X1 <-> Data Pointer/PhiSetPoints[13]
//     Term 9 (APS4322-7000)/APS Outputs/PhiE 2X2 <-> Data Pointer/PhiSetPoints[14]
//     Term 9 (APS4322-7000)/APS Outputs/PhiE 3X0 <-> Data Pointer/PhiSetPoints[18]
//     Term 9 (APS4322-7000)/APS Outputs/PhiE 3X1 <-> Data Pointer/PhiSetPoints[19]
//     Term 9 (APS4322-7000)/APS Outputs/PhiE 3X2 <-> Data Pointer/PhiSetPoints[20]
//     Term 9 (APS4322-7000)/APS Outputs/PhiE 0Y0 <-> Data Pointer/PhiSetPoints[3]
//     Term 9 (APS4322-7000)/APS Outputs/PhiE 0Y1 <-> Data Pointer/PhiSetPoints[4]
//     Term 9 (APS4322-7000)/APS Outputs/PhiE 0Y2 <-> Data Pointer/PhiSetPoints[5]
//     Term 9 (APS4322-7000)/APS Outputs/PhiE 1Y0 <-> Data Pointer/PhiSetPoints[9]
//     Term 9 (APS4322-7000)/APS Outputs/PhiE 1Y1 <-> Data Pointer/PhiSetPoints[10]
//     Term 9 (APS4322-7000)/APS Outputs/PhiE 1Y2 <-> Data Pointer/PhiSetPoints[11]
//     Term 9 (APS4322-7000)/APS Outputs/PhiE 2Y0 <-> Data Pointer/PhiSetPoints[15]
//     Term 9 (APS4322-7000)/APS Outputs/PhiE 2Y1 <-> Data Pointer/PhiSetPoints[16]
//     Term 9 (APS4322-7000)/APS Outputs/PhiE 2Y2 <-> Data Pointer/PhiSetPoints[17]
//     Term 9 (APS4322-7000)/APS Outputs/PhiE 3Y0 <-> Data Pointer/PhiSetPoints[21]
//     Term 9 (APS4322-7000)/APS Outputs/PhiE 3Y1 <-> Data Pointer/PhiSetPoints[22]
//     Term 9 (APS4322-7000)/APS Outputs/PhiE 3Y2 <-> Data Pointer/PhiSetPoints[23]
//     Term 9 (APS4322-7000)/Term 10 (APS4322-5000)/FB Inputs/A{0..8 step 2} X-Field <-> Data Pointer/HallSensorFieldsXYZ[{0..12 step 3}]  (5 links)
//     Term 9 (APS4322-7000)/Term 10 (APS4322-5000)/FB Inputs/A{0..8 step 2} Y-Field <-> Data Pointer/HallSensorFieldsXYZ[{1..13 step 3}]  (5 links)
//     Term 9 (APS4322-7000)/Term 10 (APS4322-5000)/FB Inputs/A{0..8 step 2} Z-Field <-> Data Pointer/HallSensorFieldsXYZ[{2..14 step 3}]  (5 links)
//     Term 9 (APS4322-7000)/Term 10 (APS4322-5000)/FB Inputs/B{1..9 step 2} X-Field <-> Data Pointer/HallSensorFieldsXYZ[{15..27 step 3}]  (5 links)
//     Term 9 (APS4322-7000)/Term 10 (APS4322-5000)/FB Inputs/B{1..9 step 2} Y-Field <-> Data Pointer/HallSensorFieldsXYZ[{16..28 step 3}]  (5 links)
//     Term 9 (APS4322-7000)/Term 10 (APS4322-5000)/FB Inputs/B{1..9 step 2} Z-Field <-> Data Pointer/HallSensorFieldsXYZ[{17..29 step 3}]  (5 links)
//     Term 9 (APS4322-7000)/Term 10 (APS4322-5000)/FB Inputs/C{0..8 step 2} X-Field <-> Data Pointer/HallSensorFieldsXYZ[{30..42 step 3}]  (5 links)
//     Term 9 (APS4322-7000)/Term 10 (APS4322-5000)/FB Inputs/C{0..8 step 2} Y-Field <-> Data Pointer/HallSensorFieldsXYZ[{31..43 step 3}]  (5 links)
//     Term 9 (APS4322-7000)/Term 10 (APS4322-5000)/FB Inputs/C{0..8 step 2} Z-Field <-> Data Pointer/HallSensorFieldsXYZ[{32..44 step 3}]  (5 links)
//     Term 9 (APS4322-7000)/Term 10 (APS4322-5000)/FB Inputs/D{1..9 step 2} X-Field <-> Data Pointer/HallSensorFieldsXYZ[{45..57 step 3}]  (5 links)
//     Term 9 (APS4322-7000)/Term 10 (APS4322-5000)/FB Inputs/D{1..9 step 2} Y-Field <-> Data Pointer/HallSensorFieldsXYZ[{46..58 step 3}]  (5 links)
//     Term 9 (APS4322-7000)/Term 10 (APS4322-5000)/FB Inputs/D{1..9 step 2} Z-Field <-> Data Pointer/HallSensorFieldsXYZ[{47..59 step 3}]  (5 links)
//     Term 9 (APS4322-7000)/Term 10 (APS4322-5000)/FB Inputs/E{0..8 step 2} X-Field <-> Data Pointer/HallSensorFieldsXYZ[{60..72 step 3}]  (5 links)
//     Term 9 (APS4322-7000)/Term 10 (APS4322-5000)/FB Inputs/E{0..8 step 2} Y-Field <-> Data Pointer/HallSensorFieldsXYZ[{61..73 step 3}]  (5 links)
//     Term 9 (APS4322-7000)/Term 10 (APS4322-5000)/FB Inputs/E{0..8 step 2} Z-Field <-> Data Pointer/HallSensorFieldsXYZ[{62..74 step 3}]  (5 links)
//     Term 9 (APS4322-7000)/Term 10 (APS4322-5000)/FB Inputs/F{1..9 step 2} X-Field <-> Data Pointer/HallSensorFieldsXYZ[{75..87 step 3}]  (5 links)
//     Term 9 (APS4322-7000)/Term 10 (APS4322-5000)/FB Inputs/F{1..9 step 2} Y-Field <-> Data Pointer/HallSensorFieldsXYZ[{76..88 step 3}]  (5 links)
//     Term 9 (APS4322-7000)/Term 10 (APS4322-5000)/FB Inputs/F{1..9 step 2} Z-Field <-> Data Pointer/HallSensorFieldsXYZ[{77..89 step 3}]  (5 links)
//     Term 9 (APS4322-7000)/Term 10 (APS4322-5000)/FB Inputs/G{0..8 step 2} X-Field <-> Data Pointer/HallSensorFieldsXYZ[{90..102 step 3}]  (5 links)
//     Term 9 (APS4322-7000)/Term 10 (APS4322-5000)/FB Inputs/G{0..8 step 2} Y-Field <-> Data Pointer/HallSensorFieldsXYZ[{91..103 step 3}]  (5 links)
//     Term 9 (APS4322-7000)/Term 10 (APS4322-5000)/FB Inputs/G{0..8 step 2} Z-Field <-> Data Pointer/HallSensorFieldsXYZ[{92..104 step 3}]  (5 links)
//     Term 9 (APS4322-7000)/Term 10 (APS4322-5000)/FB Inputs/H{1..9 step 2} X-Field <-> Data Pointer/HallSensorFieldsXYZ[{105..117 step 3}]  (5 links)
//     Term 9 (APS4322-7000)/Term 10 (APS4322-5000)/FB Inputs/H{1..9 step 2} Y-Field <-> Data Pointer/HallSensorFieldsXYZ[{106..118 step 3}]  (5 links)
//     Term 9 (APS4322-7000)/Term 10 (APS4322-5000)/FB Inputs/H{1..9 step 2} Z-Field <-> Data Pointer/HallSensorFieldsXYZ[{107..119 step 3}]  (5 links)
//     Term 9 (APS4322-7000)/Term 10 (APS4322-5000)/FB Inputs/I{0..8 step 2} X-Field <-> Data Pointer/HallSensorFieldsXYZ[{120..132 step 3}]  (5 links)
//     Term 9 (APS4322-7000)/Term 10 (APS4322-5000)/FB Inputs/I{0..8 step 2} Y-Field <-> Data Pointer/HallSensorFieldsXYZ[{121..133 step 3}]  (5 links)
//     Term 9 (APS4322-7000)/Term 10 (APS4322-5000)/FB Inputs/I{0..8 step 2} Z-Field <-> Data Pointer/HallSensorFieldsXYZ[{122..134 step 3}]  (5 links)
//     Term 9 (APS4322-7000)/Term 10 (APS4322-5000)/FB Inputs/J{1..9 step 2} X-Field <-> Data Pointer/HallSensorFieldsXYZ[{135..147 step 3}]  (5 links)
//     Term 9 (APS4322-7000)/Term 10 (APS4322-5000)/FB Inputs/J{1..9 step 2} Y-Field <-> Data Pointer/HallSensorFieldsXYZ[{136..148 step 3}]  (5 links)
//     Term 9 (APS4322-7000)/Term 10 (APS4322-5000)/FB Inputs/J{1..9 step 2} Z-Field <-> Data Pointer/HallSensorFieldsXYZ[{137..149 step 3}]  (5 links)
//     Term 9 (APS4322-7000)/Term 10 (APS4322-5000)/FB Inputs/Status <-> Data Pointer/FeedbackStatus
//   Device 4 (EtherCAT) <-> TcCOM Objects/XPlanar/Part1/Tile4
//     Term 11 (APS4322-7000)/APS Comm Inputs/CommStatusWord <-> Data Pointer/MoverCommStatusWord
//     Term 11 (APS4322-7000)/APS Comm Inputs/Data {1..4} <-> Data Pointer/MoverCommDataIn[{0..3}]  (4 links)
//     Term 11 (APS4322-7000)/APS Comm Outputs/CommControlWord <-> Data Pointer/MoverCommControlWord
//     Term 11 (APS4322-7000)/APS Comm Outputs/Data 1 <-> Data Pointer/MoverCommDataOut
//     Term 11 (APS4322-7000)/APS Diagdata/DC Link Voltage <-> Data Pointer/DcLinkVoltage
//     Term 11 (APS4322-7000)/APS Diagdata/Power supply current <-> Data Pointer/PowerSupplyCurrent
//     Term 11 (APS4322-7000)/APS Inputs/StatusWord <-> Data Pointer/PowerUnitStatusWord
//     Term 11 (APS4322-7000)/APS Outputs/ControlWord <-> Data Pointer/PowerUnitControlWord
//     Term 11 (APS4322-7000)/APS Outputs/Current D 0X0 <-> Data Pointer/DCurrentSetPoints[0]
//     Term 11 (APS4322-7000)/APS Outputs/Current D 0X1 <-> Data Pointer/DCurrentSetPoints[1]
//     Term 11 (APS4322-7000)/APS Outputs/Current D 0X2 <-> Data Pointer/DCurrentSetPoints[2]
//     Term 11 (APS4322-7000)/APS Outputs/Current D 1X0 <-> Data Pointer/DCurrentSetPoints[6]
//     Term 11 (APS4322-7000)/APS Outputs/Current D 1X1 <-> Data Pointer/DCurrentSetPoints[7]
//     Term 11 (APS4322-7000)/APS Outputs/Current D 1X2 <-> Data Pointer/DCurrentSetPoints[8]
//     Term 11 (APS4322-7000)/APS Outputs/Current D 2X0 <-> Data Pointer/DCurrentSetPoints[12]
//     Term 11 (APS4322-7000)/APS Outputs/Current D 2X1 <-> Data Pointer/DCurrentSetPoints[13]
//     Term 11 (APS4322-7000)/APS Outputs/Current D 2X2 <-> Data Pointer/DCurrentSetPoints[14]
//     Term 11 (APS4322-7000)/APS Outputs/Current D 3X0 <-> Data Pointer/DCurrentSetPoints[18]
//     Term 11 (APS4322-7000)/APS Outputs/Current D 3X1 <-> Data Pointer/DCurrentSetPoints[19]
//     Term 11 (APS4322-7000)/APS Outputs/Current D 3X2 <-> Data Pointer/DCurrentSetPoints[20]
//     Term 11 (APS4322-7000)/APS Outputs/Current D 0Y0 <-> Data Pointer/DCurrentSetPoints[3]
//     Term 11 (APS4322-7000)/APS Outputs/Current D 0Y1 <-> Data Pointer/DCurrentSetPoints[4]
//     Term 11 (APS4322-7000)/APS Outputs/Current D 0Y2 <-> Data Pointer/DCurrentSetPoints[5]
//     Term 11 (APS4322-7000)/APS Outputs/Current D 1Y0 <-> Data Pointer/DCurrentSetPoints[9]
//     Term 11 (APS4322-7000)/APS Outputs/Current D 1Y1 <-> Data Pointer/DCurrentSetPoints[10]
//     Term 11 (APS4322-7000)/APS Outputs/Current D 1Y2 <-> Data Pointer/DCurrentSetPoints[11]
//     Term 11 (APS4322-7000)/APS Outputs/Current D 2Y0 <-> Data Pointer/DCurrentSetPoints[15]
//     Term 11 (APS4322-7000)/APS Outputs/Current D 2Y1 <-> Data Pointer/DCurrentSetPoints[16]
//     Term 11 (APS4322-7000)/APS Outputs/Current D 2Y2 <-> Data Pointer/DCurrentSetPoints[17]
//     Term 11 (APS4322-7000)/APS Outputs/Current D 3Y0 <-> Data Pointer/DCurrentSetPoints[21]
//     Term 11 (APS4322-7000)/APS Outputs/Current D 3Y1 <-> Data Pointer/DCurrentSetPoints[22]
//     Term 11 (APS4322-7000)/APS Outputs/Current D 3Y2 <-> Data Pointer/DCurrentSetPoints[23]
//     Term 11 (APS4322-7000)/APS Outputs/Current Q 0X0 <-> Data Pointer/QCurrentSetPoints[0]
//     Term 11 (APS4322-7000)/APS Outputs/Current Q 0X1 <-> Data Pointer/QCurrentSetPoints[1]
//     Term 11 (APS4322-7000)/APS Outputs/Current Q 0X2 <-> Data Pointer/QCurrentSetPoints[2]
//     Term 11 (APS4322-7000)/APS Outputs/Current Q 1X0 <-> Data Pointer/QCurrentSetPoints[6]
//     Term 11 (APS4322-7000)/APS Outputs/Current Q 1X1 <-> Data Pointer/QCurrentSetPoints[7]
//     Term 11 (APS4322-7000)/APS Outputs/Current Q 1X2 <-> Data Pointer/QCurrentSetPoints[8]
//     Term 11 (APS4322-7000)/APS Outputs/Current Q 2X0 <-> Data Pointer/QCurrentSetPoints[12]
//     Term 11 (APS4322-7000)/APS Outputs/Current Q 2X1 <-> Data Pointer/QCurrentSetPoints[13]
//     Term 11 (APS4322-7000)/APS Outputs/Current Q 2X2 <-> Data Pointer/QCurrentSetPoints[14]
//     Term 11 (APS4322-7000)/APS Outputs/Current Q 3X0 <-> Data Pointer/QCurrentSetPoints[18]
//     Term 11 (APS4322-7000)/APS Outputs/Current Q 3X1 <-> Data Pointer/QCurrentSetPoints[19]
//     Term 11 (APS4322-7000)/APS Outputs/Current Q 3X2 <-> Data Pointer/QCurrentSetPoints[20]
//     Term 11 (APS4322-7000)/APS Outputs/Current Q 0Y0 <-> Data Pointer/QCurrentSetPoints[3]
//     Term 11 (APS4322-7000)/APS Outputs/Current Q 0Y1 <-> Data Pointer/QCurrentSetPoints[4]
//     Term 11 (APS4322-7000)/APS Outputs/Current Q 0Y2 <-> Data Pointer/QCurrentSetPoints[5]
//     Term 11 (APS4322-7000)/APS Outputs/Current Q 1Y0 <-> Data Pointer/QCurrentSetPoints[9]
//     Term 11 (APS4322-7000)/APS Outputs/Current Q 1Y1 <-> Data Pointer/QCurrentSetPoints[10]
//     Term 11 (APS4322-7000)/APS Outputs/Current Q 1Y2 <-> Data Pointer/QCurrentSetPoints[11]
//     Term 11 (APS4322-7000)/APS Outputs/Current Q 2Y0 <-> Data Pointer/QCurrentSetPoints[15]
//     Term 11 (APS4322-7000)/APS Outputs/Current Q 2Y1 <-> Data Pointer/QCurrentSetPoints[16]
//     Term 11 (APS4322-7000)/APS Outputs/Current Q 2Y2 <-> Data Pointer/QCurrentSetPoints[17]
//     Term 11 (APS4322-7000)/APS Outputs/Current Q 3Y0 <-> Data Pointer/QCurrentSetPoints[21]
//     Term 11 (APS4322-7000)/APS Outputs/Current Q 3Y1 <-> Data Pointer/QCurrentSetPoints[22]
//     Term 11 (APS4322-7000)/APS Outputs/Current Q 3Y2 <-> Data Pointer/QCurrentSetPoints[23]
//     Term 11 (APS4322-7000)/APS Outputs/PhiE 0X0 <-> Data Pointer/PhiSetPoints[0]
//     Term 11 (APS4322-7000)/APS Outputs/PhiE 0X1 <-> Data Pointer/PhiSetPoints[1]
//     Term 11 (APS4322-7000)/APS Outputs/PhiE 0X2 <-> Data Pointer/PhiSetPoints[2]
//     Term 11 (APS4322-7000)/APS Outputs/PhiE 1X0 <-> Data Pointer/PhiSetPoints[6]
//     Term 11 (APS4322-7000)/APS Outputs/PhiE 1X1 <-> Data Pointer/PhiSetPoints[7]
//     Term 11 (APS4322-7000)/APS Outputs/PhiE 1X2 <-> Data Pointer/PhiSetPoints[8]
//     Term 11 (APS4322-7000)/APS Outputs/PhiE 2X0 <-> Data Pointer/PhiSetPoints[12]
//     Term 11 (APS4322-7000)/APS Outputs/PhiE 2X1 <-> Data Pointer/PhiSetPoints[13]
//     Term 11 (APS4322-7000)/APS Outputs/PhiE 2X2 <-> Data Pointer/PhiSetPoints[14]
//     Term 11 (APS4322-7000)/APS Outputs/PhiE 3X0 <-> Data Pointer/PhiSetPoints[18]
//     Term 11 (APS4322-7000)/APS Outputs/PhiE 3X1 <-> Data Pointer/PhiSetPoints[19]
//     Term 11 (APS4322-7000)/APS Outputs/PhiE 3X2 <-> Data Pointer/PhiSetPoints[20]
//     Term 11 (APS4322-7000)/APS Outputs/PhiE 0Y0 <-> Data Pointer/PhiSetPoints[3]
//     Term 11 (APS4322-7000)/APS Outputs/PhiE 0Y1 <-> Data Pointer/PhiSetPoints[4]
//     Term 11 (APS4322-7000)/APS Outputs/PhiE 0Y2 <-> Data Pointer/PhiSetPoints[5]
//     Term 11 (APS4322-7000)/APS Outputs/PhiE 1Y0 <-> Data Pointer/PhiSetPoints[9]
//     Term 11 (APS4322-7000)/APS Outputs/PhiE 1Y1 <-> Data Pointer/PhiSetPoints[10]
//     Term 11 (APS4322-7000)/APS Outputs/PhiE 1Y2 <-> Data Pointer/PhiSetPoints[11]
//     Term 11 (APS4322-7000)/APS Outputs/PhiE 2Y0 <-> Data Pointer/PhiSetPoints[15]
//     Term 11 (APS4322-7000)/APS Outputs/PhiE 2Y1 <-> Data Pointer/PhiSetPoints[16]
//     Term 11 (APS4322-7000)/APS Outputs/PhiE 2Y2 <-> Data Pointer/PhiSetPoints[17]
//     Term 11 (APS4322-7000)/APS Outputs/PhiE 3Y0 <-> Data Pointer/PhiSetPoints[21]
//     Term 11 (APS4322-7000)/APS Outputs/PhiE 3Y1 <-> Data Pointer/PhiSetPoints[22]
//     Term 11 (APS4322-7000)/APS Outputs/PhiE 3Y2 <-> Data Pointer/PhiSetPoints[23]
//     Term 11 (APS4322-7000)/Term 12 (APS4322-5000)/FB Inputs/A{0..8 step 2} X-Field <-> Data Pointer/HallSensorFieldsXYZ[{0..12 step 3}]  (5 links)
//     Term 11 (APS4322-7000)/Term 12 (APS4322-5000)/FB Inputs/A{0..8 step 2} Y-Field <-> Data Pointer/HallSensorFieldsXYZ[{1..13 step 3}]  (5 links)
//     Term 11 (APS4322-7000)/Term 12 (APS4322-5000)/FB Inputs/A{0..8 step 2} Z-Field <-> Data Pointer/HallSensorFieldsXYZ[{2..14 step 3}]  (5 links)
//     Term 11 (APS4322-7000)/Term 12 (APS4322-5000)/FB Inputs/B{1..9 step 2} X-Field <-> Data Pointer/HallSensorFieldsXYZ[{15..27 step 3}]  (5 links)
//     Term 11 (APS4322-7000)/Term 12 (APS4322-5000)/FB Inputs/B{1..9 step 2} Y-Field <-> Data Pointer/HallSensorFieldsXYZ[{16..28 step 3}]  (5 links)
//     Term 11 (APS4322-7000)/Term 12 (APS4322-5000)/FB Inputs/B{1..9 step 2} Z-Field <-> Data Pointer/HallSensorFieldsXYZ[{17..29 step 3}]  (5 links)
//     Term 11 (APS4322-7000)/Term 12 (APS4322-5000)/FB Inputs/C{0..8 step 2} X-Field <-> Data Pointer/HallSensorFieldsXYZ[{30..42 step 3}]  (5 links)
//     Term 11 (APS4322-7000)/Term 12 (APS4322-5000)/FB Inputs/C{0..8 step 2} Y-Field <-> Data Pointer/HallSensorFieldsXYZ[{31..43 step 3}]  (5 links)
//     Term 11 (APS4322-7000)/Term 12 (APS4322-5000)/FB Inputs/C{0..8 step 2} Z-Field <-> Data Pointer/HallSensorFieldsXYZ[{32..44 step 3}]  (5 links)
//     Term 11 (APS4322-7000)/Term 12 (APS4322-5000)/FB Inputs/D{1..9 step 2} X-Field <-> Data Pointer/HallSensorFieldsXYZ[{45..57 step 3}]  (5 links)
//     Term 11 (APS4322-7000)/Term 12 (APS4322-5000)/FB Inputs/D{1..9 step 2} Y-Field <-> Data Pointer/HallSensorFieldsXYZ[{46..58 step 3}]  (5 links)
//     Term 11 (APS4322-7000)/Term 12 (APS4322-5000)/FB Inputs/D{1..9 step 2} Z-Field <-> Data Pointer/HallSensorFieldsXYZ[{47..59 step 3}]  (5 links)
//     Term 11 (APS4322-7000)/Term 12 (APS4322-5000)/FB Inputs/E{0..8 step 2} X-Field <-> Data Pointer/HallSensorFieldsXYZ[{60..72 step 3}]  (5 links)
//     Term 11 (APS4322-7000)/Term 12 (APS4322-5000)/FB Inputs/E{0..8 step 2} Y-Field <-> Data Pointer/HallSensorFieldsXYZ[{61..73 step 3}]  (5 links)
//     Term 11 (APS4322-7000)/Term 12 (APS4322-5000)/FB Inputs/E{0..8 step 2} Z-Field <-> Data Pointer/HallSensorFieldsXYZ[{62..74 step 3}]  (5 links)
//     Term 11 (APS4322-7000)/Term 12 (APS4322-5000)/FB Inputs/F{1..9 step 2} X-Field <-> Data Pointer/HallSensorFieldsXYZ[{75..87 step 3}]  (5 links)
//     Term 11 (APS4322-7000)/Term 12 (APS4322-5000)/FB Inputs/F{1..9 step 2} Y-Field <-> Data Pointer/HallSensorFieldsXYZ[{76..88 step 3}]  (5 links)
//     Term 11 (APS4322-7000)/Term 12 (APS4322-5000)/FB Inputs/F{1..9 step 2} Z-Field <-> Data Pointer/HallSensorFieldsXYZ[{77..89 step 3}]  (5 links)
//     Term 11 (APS4322-7000)/Term 12 (APS4322-5000)/FB Inputs/G{0..8 step 2} X-Field <-> Data Pointer/HallSensorFieldsXYZ[{90..102 step 3}]  (5 links)
//     Term 11 (APS4322-7000)/Term 12 (APS4322-5000)/FB Inputs/G{0..8 step 2} Y-Field <-> Data Pointer/HallSensorFieldsXYZ[{91..103 step 3}]  (5 links)
//     Term 11 (APS4322-7000)/Term 12 (APS4322-5000)/FB Inputs/G{0..8 step 2} Z-Field <-> Data Pointer/HallSensorFieldsXYZ[{92..104 step 3}]  (5 links)
//     Term 11 (APS4322-7000)/Term 12 (APS4322-5000)/FB Inputs/H{1..9 step 2} X-Field <-> Data Pointer/HallSensorFieldsXYZ[{105..117 step 3}]  (5 links)
//     Term 11 (APS4322-7000)/Term 12 (APS4322-5000)/FB Inputs/H{1..9 step 2} Y-Field <-> Data Pointer/HallSensorFieldsXYZ[{106..118 step 3}]  (5 links)
//     Term 11 (APS4322-7000)/Term 12 (APS4322-5000)/FB Inputs/H{1..9 step 2} Z-Field <-> Data Pointer/HallSensorFieldsXYZ[{107..119 step 3}]  (5 links)
//     Term 11 (APS4322-7000)/Term 12 (APS4322-5000)/FB Inputs/I{0..8 step 2} X-Field <-> Data Pointer/HallSensorFieldsXYZ[{120..132 step 3}]  (5 links)
//     Term 11 (APS4322-7000)/Term 12 (APS4322-5000)/FB Inputs/I{0..8 step 2} Y-Field <-> Data Pointer/HallSensorFieldsXYZ[{121..133 step 3}]  (5 links)
//     Term 11 (APS4322-7000)/Term 12 (APS4322-5000)/FB Inputs/I{0..8 step 2} Z-Field <-> Data Pointer/HallSensorFieldsXYZ[{122..134 step 3}]  (5 links)
//     Term 11 (APS4322-7000)/Term 12 (APS4322-5000)/FB Inputs/J{1..9 step 2} X-Field <-> Data Pointer/HallSensorFieldsXYZ[{135..147 step 3}]  (5 links)
//     Term 11 (APS4322-7000)/Term 12 (APS4322-5000)/FB Inputs/J{1..9 step 2} Y-Field <-> Data Pointer/HallSensorFieldsXYZ[{136..148 step 3}]  (5 links)
//     Term 11 (APS4322-7000)/Term 12 (APS4322-5000)/FB Inputs/J{1..9 step 2} Z-Field <-> Data Pointer/HallSensorFieldsXYZ[{137..149 step 3}]  (5 links)
//     Term 11 (APS4322-7000)/Term 12 (APS4322-5000)/FB Inputs/Status <-> Data Pointer/FeedbackStatus
//   Device 4 (EtherCAT) <-> TcCOM Objects/XPlanar/Part1/Tile5
//     Term 13 (APS4322-7000)/APS Comm Inputs/CommStatusWord <-> Data Pointer/MoverCommStatusWord
//     Term 13 (APS4322-7000)/APS Comm Inputs/Data {1..4} <-> Data Pointer/MoverCommDataIn[{0..3}]  (4 links)
//     Term 13 (APS4322-7000)/APS Comm Outputs/CommControlWord <-> Data Pointer/MoverCommControlWord
//     Term 13 (APS4322-7000)/APS Comm Outputs/Data 1 <-> Data Pointer/MoverCommDataOut
//     Term 13 (APS4322-7000)/APS Diagdata/DC Link Voltage <-> Data Pointer/DcLinkVoltage
//     Term 13 (APS4322-7000)/APS Diagdata/Power supply current <-> Data Pointer/PowerSupplyCurrent
//     Term 13 (APS4322-7000)/APS Inputs/StatusWord <-> Data Pointer/PowerUnitStatusWord
//     Term 13 (APS4322-7000)/APS Outputs/ControlWord <-> Data Pointer/PowerUnitControlWord
//     Term 13 (APS4322-7000)/APS Outputs/Current D 0X0 <-> Data Pointer/DCurrentSetPoints[0]
//     Term 13 (APS4322-7000)/APS Outputs/Current D 0X1 <-> Data Pointer/DCurrentSetPoints[1]
//     Term 13 (APS4322-7000)/APS Outputs/Current D 0X2 <-> Data Pointer/DCurrentSetPoints[2]
//     Term 13 (APS4322-7000)/APS Outputs/Current D 1X0 <-> Data Pointer/DCurrentSetPoints[6]
//     Term 13 (APS4322-7000)/APS Outputs/Current D 1X1 <-> Data Pointer/DCurrentSetPoints[7]
//     Term 13 (APS4322-7000)/APS Outputs/Current D 1X2 <-> Data Pointer/DCurrentSetPoints[8]
//     Term 13 (APS4322-7000)/APS Outputs/Current D 2X0 <-> Data Pointer/DCurrentSetPoints[12]
//     Term 13 (APS4322-7000)/APS Outputs/Current D 2X1 <-> Data Pointer/DCurrentSetPoints[13]
//     Term 13 (APS4322-7000)/APS Outputs/Current D 2X2 <-> Data Pointer/DCurrentSetPoints[14]
//     Term 13 (APS4322-7000)/APS Outputs/Current D 3X0 <-> Data Pointer/DCurrentSetPoints[18]
//     Term 13 (APS4322-7000)/APS Outputs/Current D 3X1 <-> Data Pointer/DCurrentSetPoints[19]
//     Term 13 (APS4322-7000)/APS Outputs/Current D 3X2 <-> Data Pointer/DCurrentSetPoints[20]
//     Term 13 (APS4322-7000)/APS Outputs/Current D 0Y0 <-> Data Pointer/DCurrentSetPoints[3]
//     Term 13 (APS4322-7000)/APS Outputs/Current D 0Y1 <-> Data Pointer/DCurrentSetPoints[4]
//     Term 13 (APS4322-7000)/APS Outputs/Current D 0Y2 <-> Data Pointer/DCurrentSetPoints[5]
//     Term 13 (APS4322-7000)/APS Outputs/Current D 1Y0 <-> Data Pointer/DCurrentSetPoints[9]
//     Term 13 (APS4322-7000)/APS Outputs/Current D 1Y1 <-> Data Pointer/DCurrentSetPoints[10]
//     Term 13 (APS4322-7000)/APS Outputs/Current D 1Y2 <-> Data Pointer/DCurrentSetPoints[11]
//     Term 13 (APS4322-7000)/APS Outputs/Current D 2Y0 <-> Data Pointer/DCurrentSetPoints[15]
//     Term 13 (APS4322-7000)/APS Outputs/Current D 2Y1 <-> Data Pointer/DCurrentSetPoints[16]
//     Term 13 (APS4322-7000)/APS Outputs/Current D 2Y2 <-> Data Pointer/DCurrentSetPoints[17]
//     Term 13 (APS4322-7000)/APS Outputs/Current D 3Y0 <-> Data Pointer/DCurrentSetPoints[21]
//     Term 13 (APS4322-7000)/APS Outputs/Current D 3Y1 <-> Data Pointer/DCurrentSetPoints[22]
//     Term 13 (APS4322-7000)/APS Outputs/Current D 3Y2 <-> Data Pointer/DCurrentSetPoints[23]
//     Term 13 (APS4322-7000)/APS Outputs/Current Q 0X0 <-> Data Pointer/QCurrentSetPoints[0]
//     Term 13 (APS4322-7000)/APS Outputs/Current Q 0X1 <-> Data Pointer/QCurrentSetPoints[1]
//     Term 13 (APS4322-7000)/APS Outputs/Current Q 0X2 <-> Data Pointer/QCurrentSetPoints[2]
//     Term 13 (APS4322-7000)/APS Outputs/Current Q 1X0 <-> Data Pointer/QCurrentSetPoints[6]
//     Term 13 (APS4322-7000)/APS Outputs/Current Q 1X1 <-> Data Pointer/QCurrentSetPoints[7]
//     Term 13 (APS4322-7000)/APS Outputs/Current Q 1X2 <-> Data Pointer/QCurrentSetPoints[8]
//     Term 13 (APS4322-7000)/APS Outputs/Current Q 2X0 <-> Data Pointer/QCurrentSetPoints[12]
//     Term 13 (APS4322-7000)/APS Outputs/Current Q 2X1 <-> Data Pointer/QCurrentSetPoints[13]
//     Term 13 (APS4322-7000)/APS Outputs/Current Q 2X2 <-> Data Pointer/QCurrentSetPoints[14]
//     Term 13 (APS4322-7000)/APS Outputs/Current Q 3X0 <-> Data Pointer/QCurrentSetPoints[18]
//     Term 13 (APS4322-7000)/APS Outputs/Current Q 3X1 <-> Data Pointer/QCurrentSetPoints[19]
//     Term 13 (APS4322-7000)/APS Outputs/Current Q 3X2 <-> Data Pointer/QCurrentSetPoints[20]
//     Term 13 (APS4322-7000)/APS Outputs/Current Q 0Y0 <-> Data Pointer/QCurrentSetPoints[3]
//     Term 13 (APS4322-7000)/APS Outputs/Current Q 0Y1 <-> Data Pointer/QCurrentSetPoints[4]
//     Term 13 (APS4322-7000)/APS Outputs/Current Q 0Y2 <-> Data Pointer/QCurrentSetPoints[5]
//     Term 13 (APS4322-7000)/APS Outputs/Current Q 1Y0 <-> Data Pointer/QCurrentSetPoints[9]
//     Term 13 (APS4322-7000)/APS Outputs/Current Q 1Y1 <-> Data Pointer/QCurrentSetPoints[10]
//     Term 13 (APS4322-7000)/APS Outputs/Current Q 1Y2 <-> Data Pointer/QCurrentSetPoints[11]
//     Term 13 (APS4322-7000)/APS Outputs/Current Q 2Y0 <-> Data Pointer/QCurrentSetPoints[15]
//     Term 13 (APS4322-7000)/APS Outputs/Current Q 2Y1 <-> Data Pointer/QCurrentSetPoints[16]
//     Term 13 (APS4322-7000)/APS Outputs/Current Q 2Y2 <-> Data Pointer/QCurrentSetPoints[17]
//     Term 13 (APS4322-7000)/APS Outputs/Current Q 3Y0 <-> Data Pointer/QCurrentSetPoints[21]
//     Term 13 (APS4322-7000)/APS Outputs/Current Q 3Y1 <-> Data Pointer/QCurrentSetPoints[22]
//     Term 13 (APS4322-7000)/APS Outputs/Current Q 3Y2 <-> Data Pointer/QCurrentSetPoints[23]
//     Term 13 (APS4322-7000)/APS Outputs/PhiE 0X0 <-> Data Pointer/PhiSetPoints[0]
//     Term 13 (APS4322-7000)/APS Outputs/PhiE 0X1 <-> Data Pointer/PhiSetPoints[1]
//     Term 13 (APS4322-7000)/APS Outputs/PhiE 0X2 <-> Data Pointer/PhiSetPoints[2]
//     Term 13 (APS4322-7000)/APS Outputs/PhiE 1X0 <-> Data Pointer/PhiSetPoints[6]
//     Term 13 (APS4322-7000)/APS Outputs/PhiE 1X1 <-> Data Pointer/PhiSetPoints[7]
//     Term 13 (APS4322-7000)/APS Outputs/PhiE 1X2 <-> Data Pointer/PhiSetPoints[8]
//     Term 13 (APS4322-7000)/APS Outputs/PhiE 2X0 <-> Data Pointer/PhiSetPoints[12]
//     Term 13 (APS4322-7000)/APS Outputs/PhiE 2X1 <-> Data Pointer/PhiSetPoints[13]
//     Term 13 (APS4322-7000)/APS Outputs/PhiE 2X2 <-> Data Pointer/PhiSetPoints[14]
//     Term 13 (APS4322-7000)/APS Outputs/PhiE 3X0 <-> Data Pointer/PhiSetPoints[18]
//     Term 13 (APS4322-7000)/APS Outputs/PhiE 3X1 <-> Data Pointer/PhiSetPoints[19]
//     Term 13 (APS4322-7000)/APS Outputs/PhiE 3X2 <-> Data Pointer/PhiSetPoints[20]
//     Term 13 (APS4322-7000)/APS Outputs/PhiE 0Y0 <-> Data Pointer/PhiSetPoints[3]
//     Term 13 (APS4322-7000)/APS Outputs/PhiE 0Y1 <-> Data Pointer/PhiSetPoints[4]
//     Term 13 (APS4322-7000)/APS Outputs/PhiE 0Y2 <-> Data Pointer/PhiSetPoints[5]
//     Term 13 (APS4322-7000)/APS Outputs/PhiE 1Y0 <-> Data Pointer/PhiSetPoints[9]
//     Term 13 (APS4322-7000)/APS Outputs/PhiE 1Y1 <-> Data Pointer/PhiSetPoints[10]
//     Term 13 (APS4322-7000)/APS Outputs/PhiE 1Y2 <-> Data Pointer/PhiSetPoints[11]
//     Term 13 (APS4322-7000)/APS Outputs/PhiE 2Y0 <-> Data Pointer/PhiSetPoints[15]
//     Term 13 (APS4322-7000)/APS Outputs/PhiE 2Y1 <-> Data Pointer/PhiSetPoints[16]
//     Term 13 (APS4322-7000)/APS Outputs/PhiE 2Y2 <-> Data Pointer/PhiSetPoints[17]
//     Term 13 (APS4322-7000)/APS Outputs/PhiE 3Y0 <-> Data Pointer/PhiSetPoints[21]
//     Term 13 (APS4322-7000)/APS Outputs/PhiE 3Y1 <-> Data Pointer/PhiSetPoints[22]
//     Term 13 (APS4322-7000)/APS Outputs/PhiE 3Y2 <-> Data Pointer/PhiSetPoints[23]
//     Term 13 (APS4322-7000)/Term 14 (APS4322-5000)/FB Inputs/A{0..8 step 2} X-Field <-> Data Pointer/HallSensorFieldsXYZ[{0..12 step 3}]  (5 links)
//     Term 13 (APS4322-7000)/Term 14 (APS4322-5000)/FB Inputs/A{0..8 step 2} Y-Field <-> Data Pointer/HallSensorFieldsXYZ[{1..13 step 3}]  (5 links)
//     Term 13 (APS4322-7000)/Term 14 (APS4322-5000)/FB Inputs/A{0..8 step 2} Z-Field <-> Data Pointer/HallSensorFieldsXYZ[{2..14 step 3}]  (5 links)
//     Term 13 (APS4322-7000)/Term 14 (APS4322-5000)/FB Inputs/B{1..9 step 2} X-Field <-> Data Pointer/HallSensorFieldsXYZ[{15..27 step 3}]  (5 links)
//     Term 13 (APS4322-7000)/Term 14 (APS4322-5000)/FB Inputs/B{1..9 step 2} Y-Field <-> Data Pointer/HallSensorFieldsXYZ[{16..28 step 3}]  (5 links)
//     Term 13 (APS4322-7000)/Term 14 (APS4322-5000)/FB Inputs/B{1..9 step 2} Z-Field <-> Data Pointer/HallSensorFieldsXYZ[{17..29 step 3}]  (5 links)
//     Term 13 (APS4322-7000)/Term 14 (APS4322-5000)/FB Inputs/C{0..8 step 2} X-Field <-> Data Pointer/HallSensorFieldsXYZ[{30..42 step 3}]  (5 links)
//     Term 13 (APS4322-7000)/Term 14 (APS4322-5000)/FB Inputs/C{0..8 step 2} Y-Field <-> Data Pointer/HallSensorFieldsXYZ[{31..43 step 3}]  (5 links)
//     Term 13 (APS4322-7000)/Term 14 (APS4322-5000)/FB Inputs/C{0..8 step 2} Z-Field <-> Data Pointer/HallSensorFieldsXYZ[{32..44 step 3}]  (5 links)
//     Term 13 (APS4322-7000)/Term 14 (APS4322-5000)/FB Inputs/D{1..9 step 2} X-Field <-> Data Pointer/HallSensorFieldsXYZ[{45..57 step 3}]  (5 links)
//     Term 13 (APS4322-7000)/Term 14 (APS4322-5000)/FB Inputs/D{1..9 step 2} Y-Field <-> Data Pointer/HallSensorFieldsXYZ[{46..58 step 3}]  (5 links)
//     Term 13 (APS4322-7000)/Term 14 (APS4322-5000)/FB Inputs/D{1..9 step 2} Z-Field <-> Data Pointer/HallSensorFieldsXYZ[{47..59 step 3}]  (5 links)
//     Term 13 (APS4322-7000)/Term 14 (APS4322-5000)/FB Inputs/E{0..8 step 2} X-Field <-> Data Pointer/HallSensorFieldsXYZ[{60..72 step 3}]  (5 links)
//     Term 13 (APS4322-7000)/Term 14 (APS4322-5000)/FB Inputs/E{0..8 step 2} Y-Field <-> Data Pointer/HallSensorFieldsXYZ[{61..73 step 3}]  (5 links)
//     Term 13 (APS4322-7000)/Term 14 (APS4322-5000)/FB Inputs/E{0..8 step 2} Z-Field <-> Data Pointer/HallSensorFieldsXYZ[{62..74 step 3}]  (5 links)
//     Term 13 (APS4322-7000)/Term 14 (APS4322-5000)/FB Inputs/F{1..9 step 2} X-Field <-> Data Pointer/HallSensorFieldsXYZ[{75..87 step 3}]  (5 links)
//     Term 13 (APS4322-7000)/Term 14 (APS4322-5000)/FB Inputs/F{1..9 step 2} Y-Field <-> Data Pointer/HallSensorFieldsXYZ[{76..88 step 3}]  (5 links)
//     Term 13 (APS4322-7000)/Term 14 (APS4322-5000)/FB Inputs/F{1..9 step 2} Z-Field <-> Data Pointer/HallSensorFieldsXYZ[{77..89 step 3}]  (5 links)
//     Term 13 (APS4322-7000)/Term 14 (APS4322-5000)/FB Inputs/G{0..8 step 2} X-Field <-> Data Pointer/HallSensorFieldsXYZ[{90..102 step 3}]  (5 links)
//     Term 13 (APS4322-7000)/Term 14 (APS4322-5000)/FB Inputs/G{0..8 step 2} Y-Field <-> Data Pointer/HallSensorFieldsXYZ[{91..103 step 3}]  (5 links)
//     Term 13 (APS4322-7000)/Term 14 (APS4322-5000)/FB Inputs/G{0..8 step 2} Z-Field <-> Data Pointer/HallSensorFieldsXYZ[{92..104 step 3}]  (5 links)
//     Term 13 (APS4322-7000)/Term 14 (APS4322-5000)/FB Inputs/H{1..9 step 2} X-Field <-> Data Pointer/HallSensorFieldsXYZ[{105..117 step 3}]  (5 links)
//     Term 13 (APS4322-7000)/Term 14 (APS4322-5000)/FB Inputs/H{1..9 step 2} Y-Field <-> Data Pointer/HallSensorFieldsXYZ[{106..118 step 3}]  (5 links)
//     Term 13 (APS4322-7000)/Term 14 (APS4322-5000)/FB Inputs/H{1..9 step 2} Z-Field <-> Data Pointer/HallSensorFieldsXYZ[{107..119 step 3}]  (5 links)
//     Term 13 (APS4322-7000)/Term 14 (APS4322-5000)/FB Inputs/I{0..8 step 2} X-Field <-> Data Pointer/HallSensorFieldsXYZ[{120..132 step 3}]  (5 links)
//     Term 13 (APS4322-7000)/Term 14 (APS4322-5000)/FB Inputs/I{0..8 step 2} Y-Field <-> Data Pointer/HallSensorFieldsXYZ[{121..133 step 3}]  (5 links)
//     Term 13 (APS4322-7000)/Term 14 (APS4322-5000)/FB Inputs/I{0..8 step 2} Z-Field <-> Data Pointer/HallSensorFieldsXYZ[{122..134 step 3}]  (5 links)
//     Term 13 (APS4322-7000)/Term 14 (APS4322-5000)/FB Inputs/J{1..9 step 2} X-Field <-> Data Pointer/HallSensorFieldsXYZ[{135..147 step 3}]  (5 links)
//     Term 13 (APS4322-7000)/Term 14 (APS4322-5000)/FB Inputs/J{1..9 step 2} Y-Field <-> Data Pointer/HallSensorFieldsXYZ[{136..148 step 3}]  (5 links)
//     Term 13 (APS4322-7000)/Term 14 (APS4322-5000)/FB Inputs/J{1..9 step 2} Z-Field <-> Data Pointer/HallSensorFieldsXYZ[{137..149 step 3}]  (5 links)
//     Term 13 (APS4322-7000)/Term 14 (APS4322-5000)/FB Inputs/Status <-> Data Pointer/FeedbackStatus
//   Device 4 (EtherCAT) <-> TcCOM Objects/XPlanar/Part1/Tile6
//     Term 15 (APS4322-7000)/APS Comm Inputs/CommStatusWord <-> Data Pointer/MoverCommStatusWord
//     Term 15 (APS4322-7000)/APS Comm Inputs/Data {1..4} <-> Data Pointer/MoverCommDataIn[{0..3}]  (4 links)
//     Term 15 (APS4322-7000)/APS Comm Outputs/CommControlWord <-> Data Pointer/MoverCommControlWord
//     Term 15 (APS4322-7000)/APS Comm Outputs/Data 1 <-> Data Pointer/MoverCommDataOut
//     Term 15 (APS4322-7000)/APS Diagdata/DC Link Voltage <-> Data Pointer/DcLinkVoltage
//     Term 15 (APS4322-7000)/APS Diagdata/Power supply current <-> Data Pointer/PowerSupplyCurrent
//     Term 15 (APS4322-7000)/APS Inputs/StatusWord <-> Data Pointer/PowerUnitStatusWord
//     Term 15 (APS4322-7000)/APS Outputs/ControlWord <-> Data Pointer/PowerUnitControlWord
//     Term 15 (APS4322-7000)/APS Outputs/Current D 0X0 <-> Data Pointer/DCurrentSetPoints[0]
//     Term 15 (APS4322-7000)/APS Outputs/Current D 0X1 <-> Data Pointer/DCurrentSetPoints[1]
//     Term 15 (APS4322-7000)/APS Outputs/Current D 0X2 <-> Data Pointer/DCurrentSetPoints[2]
//     Term 15 (APS4322-7000)/APS Outputs/Current D 1X0 <-> Data Pointer/DCurrentSetPoints[6]
//     Term 15 (APS4322-7000)/APS Outputs/Current D 1X1 <-> Data Pointer/DCurrentSetPoints[7]
//     Term 15 (APS4322-7000)/APS Outputs/Current D 1X2 <-> Data Pointer/DCurrentSetPoints[8]
//     Term 15 (APS4322-7000)/APS Outputs/Current D 2X0 <-> Data Pointer/DCurrentSetPoints[12]
//     Term 15 (APS4322-7000)/APS Outputs/Current D 2X1 <-> Data Pointer/DCurrentSetPoints[13]
//     Term 15 (APS4322-7000)/APS Outputs/Current D 2X2 <-> Data Pointer/DCurrentSetPoints[14]
//     Term 15 (APS4322-7000)/APS Outputs/Current D 3X0 <-> Data Pointer/DCurrentSetPoints[18]
//     Term 15 (APS4322-7000)/APS Outputs/Current D 3X1 <-> Data Pointer/DCurrentSetPoints[19]
//     Term 15 (APS4322-7000)/APS Outputs/Current D 3X2 <-> Data Pointer/DCurrentSetPoints[20]
//     Term 15 (APS4322-7000)/APS Outputs/Current D 0Y0 <-> Data Pointer/DCurrentSetPoints[3]
//     Term 15 (APS4322-7000)/APS Outputs/Current D 0Y1 <-> Data Pointer/DCurrentSetPoints[4]
//     Term 15 (APS4322-7000)/APS Outputs/Current D 0Y2 <-> Data Pointer/DCurrentSetPoints[5]
//     Term 15 (APS4322-7000)/APS Outputs/Current D 1Y0 <-> Data Pointer/DCurrentSetPoints[9]
//     Term 15 (APS4322-7000)/APS Outputs/Current D 1Y1 <-> Data Pointer/DCurrentSetPoints[10]
//     Term 15 (APS4322-7000)/APS Outputs/Current D 1Y2 <-> Data Pointer/DCurrentSetPoints[11]
//     Term 15 (APS4322-7000)/APS Outputs/Current D 2Y0 <-> Data Pointer/DCurrentSetPoints[15]
//     Term 15 (APS4322-7000)/APS Outputs/Current D 2Y1 <-> Data Pointer/DCurrentSetPoints[16]
//     Term 15 (APS4322-7000)/APS Outputs/Current D 2Y2 <-> Data Pointer/DCurrentSetPoints[17]
//     Term 15 (APS4322-7000)/APS Outputs/Current D 3Y0 <-> Data Pointer/DCurrentSetPoints[21]
//     Term 15 (APS4322-7000)/APS Outputs/Current D 3Y1 <-> Data Pointer/DCurrentSetPoints[22]
//     Term 15 (APS4322-7000)/APS Outputs/Current D 3Y2 <-> Data Pointer/DCurrentSetPoints[23]
//     Term 15 (APS4322-7000)/APS Outputs/Current Q 0X0 <-> Data Pointer/QCurrentSetPoints[0]
//     Term 15 (APS4322-7000)/APS Outputs/Current Q 0X1 <-> Data Pointer/QCurrentSetPoints[1]
//     Term 15 (APS4322-7000)/APS Outputs/Current Q 0X2 <-> Data Pointer/QCurrentSetPoints[2]
//     Term 15 (APS4322-7000)/APS Outputs/Current Q 1X0 <-> Data Pointer/QCurrentSetPoints[6]
//     Term 15 (APS4322-7000)/APS Outputs/Current Q 1X1 <-> Data Pointer/QCurrentSetPoints[7]
//     Term 15 (APS4322-7000)/APS Outputs/Current Q 1X2 <-> Data Pointer/QCurrentSetPoints[8]
//     Term 15 (APS4322-7000)/APS Outputs/Current Q 2X0 <-> Data Pointer/QCurrentSetPoints[12]
//     Term 15 (APS4322-7000)/APS Outputs/Current Q 2X1 <-> Data Pointer/QCurrentSetPoints[13]
//     Term 15 (APS4322-7000)/APS Outputs/Current Q 2X2 <-> Data Pointer/QCurrentSetPoints[14]
//     Term 15 (APS4322-7000)/APS Outputs/Current Q 3X0 <-> Data Pointer/QCurrentSetPoints[18]
//     Term 15 (APS4322-7000)/APS Outputs/Current Q 3X1 <-> Data Pointer/QCurrentSetPoints[19]
//     Term 15 (APS4322-7000)/APS Outputs/Current Q 3X2 <-> Data Pointer/QCurrentSetPoints[20]
//     Term 15 (APS4322-7000)/APS Outputs/Current Q 0Y0 <-> Data Pointer/QCurrentSetPoints[3]
//     Term 15 (APS4322-7000)/APS Outputs/Current Q 0Y1 <-> Data Pointer/QCurrentSetPoints[4]
//     Term 15 (APS4322-7000)/APS Outputs/Current Q 0Y2 <-> Data Pointer/QCurrentSetPoints[5]
//     Term 15 (APS4322-7000)/APS Outputs/Current Q 1Y0 <-> Data Pointer/QCurrentSetPoints[9]
//     Term 15 (APS4322-7000)/APS Outputs/Current Q 1Y1 <-> Data Pointer/QCurrentSetPoints[10]
//     Term 15 (APS4322-7000)/APS Outputs/Current Q 1Y2 <-> Data Pointer/QCurrentSetPoints[11]
//     Term 15 (APS4322-7000)/APS Outputs/Current Q 2Y0 <-> Data Pointer/QCurrentSetPoints[15]
//     Term 15 (APS4322-7000)/APS Outputs/Current Q 2Y1 <-> Data Pointer/QCurrentSetPoints[16]
//     Term 15 (APS4322-7000)/APS Outputs/Current Q 2Y2 <-> Data Pointer/QCurrentSetPoints[17]
//     Term 15 (APS4322-7000)/APS Outputs/Current Q 3Y0 <-> Data Pointer/QCurrentSetPoints[21]
//     Term 15 (APS4322-7000)/APS Outputs/Current Q 3Y1 <-> Data Pointer/QCurrentSetPoints[22]
//     Term 15 (APS4322-7000)/APS Outputs/Current Q 3Y2 <-> Data Pointer/QCurrentSetPoints[23]
//     Term 15 (APS4322-7000)/APS Outputs/PhiE 0X0 <-> Data Pointer/PhiSetPoints[0]
//     Term 15 (APS4322-7000)/APS Outputs/PhiE 0X1 <-> Data Pointer/PhiSetPoints[1]
//     Term 15 (APS4322-7000)/APS Outputs/PhiE 0X2 <-> Data Pointer/PhiSetPoints[2]
//     Term 15 (APS4322-7000)/APS Outputs/PhiE 1X0 <-> Data Pointer/PhiSetPoints[6]
//     Term 15 (APS4322-7000)/APS Outputs/PhiE 1X1 <-> Data Pointer/PhiSetPoints[7]
//     Term 15 (APS4322-7000)/APS Outputs/PhiE 1X2 <-> Data Pointer/PhiSetPoints[8]
//     Term 15 (APS4322-7000)/APS Outputs/PhiE 2X0 <-> Data Pointer/PhiSetPoints[12]
//     Term 15 (APS4322-7000)/APS Outputs/PhiE 2X1 <-> Data Pointer/PhiSetPoints[13]
//     Term 15 (APS4322-7000)/APS Outputs/PhiE 2X2 <-> Data Pointer/PhiSetPoints[14]
//     Term 15 (APS4322-7000)/APS Outputs/PhiE 3X0 <-> Data Pointer/PhiSetPoints[18]
//     Term 15 (APS4322-7000)/APS Outputs/PhiE 3X1 <-> Data Pointer/PhiSetPoints[19]
//     Term 15 (APS4322-7000)/APS Outputs/PhiE 3X2 <-> Data Pointer/PhiSetPoints[20]
//     Term 15 (APS4322-7000)/APS Outputs/PhiE 0Y0 <-> Data Pointer/PhiSetPoints[3]
//     Term 15 (APS4322-7000)/APS Outputs/PhiE 0Y1 <-> Data Pointer/PhiSetPoints[4]
//     Term 15 (APS4322-7000)/APS Outputs/PhiE 0Y2 <-> Data Pointer/PhiSetPoints[5]
//     Term 15 (APS4322-7000)/APS Outputs/PhiE 1Y0 <-> Data Pointer/PhiSetPoints[9]
//     Term 15 (APS4322-7000)/APS Outputs/PhiE 1Y1 <-> Data Pointer/PhiSetPoints[10]
//     Term 15 (APS4322-7000)/APS Outputs/PhiE 1Y2 <-> Data Pointer/PhiSetPoints[11]
//     Term 15 (APS4322-7000)/APS Outputs/PhiE 2Y0 <-> Data Pointer/PhiSetPoints[15]
//     Term 15 (APS4322-7000)/APS Outputs/PhiE 2Y1 <-> Data Pointer/PhiSetPoints[16]
//     Term 15 (APS4322-7000)/APS Outputs/PhiE 2Y2 <-> Data Pointer/PhiSetPoints[17]
//     Term 15 (APS4322-7000)/APS Outputs/PhiE 3Y0 <-> Data Pointer/PhiSetPoints[21]
//     Term 15 (APS4322-7000)/APS Outputs/PhiE 3Y1 <-> Data Pointer/PhiSetPoints[22]
//     Term 15 (APS4322-7000)/APS Outputs/PhiE 3Y2 <-> Data Pointer/PhiSetPoints[23]
//     Term 15 (APS4322-7000)/Term 16 (APS4322-5000)/FB Inputs/A{0..8 step 2} X-Field <-> Data Pointer/HallSensorFieldsXYZ[{0..12 step 3}]  (5 links)
//     Term 15 (APS4322-7000)/Term 16 (APS4322-5000)/FB Inputs/A{0..8 step 2} Y-Field <-> Data Pointer/HallSensorFieldsXYZ[{1..13 step 3}]  (5 links)
//     Term 15 (APS4322-7000)/Term 16 (APS4322-5000)/FB Inputs/A{0..8 step 2} Z-Field <-> Data Pointer/HallSensorFieldsXYZ[{2..14 step 3}]  (5 links)
//     Term 15 (APS4322-7000)/Term 16 (APS4322-5000)/FB Inputs/B{1..9 step 2} X-Field <-> Data Pointer/HallSensorFieldsXYZ[{15..27 step 3}]  (5 links)
//     Term 15 (APS4322-7000)/Term 16 (APS4322-5000)/FB Inputs/B{1..9 step 2} Y-Field <-> Data Pointer/HallSensorFieldsXYZ[{16..28 step 3}]  (5 links)
//     Term 15 (APS4322-7000)/Term 16 (APS4322-5000)/FB Inputs/B{1..9 step 2} Z-Field <-> Data Pointer/HallSensorFieldsXYZ[{17..29 step 3}]  (5 links)
//     Term 15 (APS4322-7000)/Term 16 (APS4322-5000)/FB Inputs/C{0..8 step 2} X-Field <-> Data Pointer/HallSensorFieldsXYZ[{30..42 step 3}]  (5 links)
//     Term 15 (APS4322-7000)/Term 16 (APS4322-5000)/FB Inputs/C{0..8 step 2} Y-Field <-> Data Pointer/HallSensorFieldsXYZ[{31..43 step 3}]  (5 links)
//     Term 15 (APS4322-7000)/Term 16 (APS4322-5000)/FB Inputs/C{0..8 step 2} Z-Field <-> Data Pointer/HallSensorFieldsXYZ[{32..44 step 3}]  (5 links)
//     Term 15 (APS4322-7000)/Term 16 (APS4322-5000)/FB Inputs/D{1..9 step 2} X-Field <-> Data Pointer/HallSensorFieldsXYZ[{45..57 step 3}]  (5 links)
//     Term 15 (APS4322-7000)/Term 16 (APS4322-5000)/FB Inputs/D{1..9 step 2} Y-Field <-> Data Pointer/HallSensorFieldsXYZ[{46..58 step 3}]  (5 links)
//     Term 15 (APS4322-7000)/Term 16 (APS4322-5000)/FB Inputs/D{1..9 step 2} Z-Field <-> Data Pointer/HallSensorFieldsXYZ[{47..59 step 3}]  (5 links)
//     Term 15 (APS4322-7000)/Term 16 (APS4322-5000)/FB Inputs/E{0..8 step 2} X-Field <-> Data Pointer/HallSensorFieldsXYZ[{60..72 step 3}]  (5 links)
//     Term 15 (APS4322-7000)/Term 16 (APS4322-5000)/FB Inputs/E{0..8 step 2} Y-Field <-> Data Pointer/HallSensorFieldsXYZ[{61..73 step 3}]  (5 links)
//     Term 15 (APS4322-7000)/Term 16 (APS4322-5000)/FB Inputs/E{0..8 step 2} Z-Field <-> Data Pointer/HallSensorFieldsXYZ[{62..74 step 3}]  (5 links)
//     Term 15 (APS4322-7000)/Term 16 (APS4322-5000)/FB Inputs/F{1..9 step 2} X-Field <-> Data Pointer/HallSensorFieldsXYZ[{75..87 step 3}]  (5 links)
//     Term 15 (APS4322-7000)/Term 16 (APS4322-5000)/FB Inputs/F{1..9 step 2} Y-Field <-> Data Pointer/HallSensorFieldsXYZ[{76..88 step 3}]  (5 links)
//     Term 15 (APS4322-7000)/Term 16 (APS4322-5000)/FB Inputs/F{1..9 step 2} Z-Field <-> Data Pointer/HallSensorFieldsXYZ[{77..89 step 3}]  (5 links)
//     Term 15 (APS4322-7000)/Term 16 (APS4322-5000)/FB Inputs/G{0..8 step 2} X-Field <-> Data Pointer/HallSensorFieldsXYZ[{90..102 step 3}]  (5 links)
//     Term 15 (APS4322-7000)/Term 16 (APS4322-5000)/FB Inputs/G{0..8 step 2} Y-Field <-> Data Pointer/HallSensorFieldsXYZ[{91..103 step 3}]  (5 links)
//     Term 15 (APS4322-7000)/Term 16 (APS4322-5000)/FB Inputs/G{0..8 step 2} Z-Field <-> Data Pointer/HallSensorFieldsXYZ[{92..104 step 3}]  (5 links)
//     Term 15 (APS4322-7000)/Term 16 (APS4322-5000)/FB Inputs/H{1..9 step 2} X-Field <-> Data Pointer/HallSensorFieldsXYZ[{105..117 step 3}]  (5 links)
//     Term 15 (APS4322-7000)/Term 16 (APS4322-5000)/FB Inputs/H{1..9 step 2} Y-Field <-> Data Pointer/HallSensorFieldsXYZ[{106..118 step 3}]  (5 links)
//     Term 15 (APS4322-7000)/Term 16 (APS4322-5000)/FB Inputs/H{1..9 step 2} Z-Field <-> Data Pointer/HallSensorFieldsXYZ[{107..119 step 3}]  (5 links)
//     Term 15 (APS4322-7000)/Term 16 (APS4322-5000)/FB Inputs/I{0..8 step 2} X-Field <-> Data Pointer/HallSensorFieldsXYZ[{120..132 step 3}]  (5 links)
//     Term 15 (APS4322-7000)/Term 16 (APS4322-5000)/FB Inputs/I{0..8 step 2} Y-Field <-> Data Pointer/HallSensorFieldsXYZ[{121..133 step 3}]  (5 links)
//     Term 15 (APS4322-7000)/Term 16 (APS4322-5000)/FB Inputs/I{0..8 step 2} Z-Field <-> Data Pointer/HallSensorFieldsXYZ[{122..134 step 3}]  (5 links)
//     Term 15 (APS4322-7000)/Term 16 (APS4322-5000)/FB Inputs/J{1..9 step 2} X-Field <-> Data Pointer/HallSensorFieldsXYZ[{135..147 step 3}]  (5 links)
//     Term 15 (APS4322-7000)/Term 16 (APS4322-5000)/FB Inputs/J{1..9 step 2} Y-Field <-> Data Pointer/HallSensorFieldsXYZ[{136..148 step 3}]  (5 links)
//     Term 15 (APS4322-7000)/Term 16 (APS4322-5000)/FB Inputs/J{1..9 step 2} Z-Field <-> Data Pointer/HallSensorFieldsXYZ[{137..149 step 3}]  (5 links)
//     Term 15 (APS4322-7000)/Term 16 (APS4322-5000)/FB Inputs/Status <-> Data Pointer/FeedbackStatus
//   XPlanar MC Project/Axes/Mover4220_1 <-> TcCOM Objects/XPlanar/Mover4220_1
//     IoToMc/STD <-> OutputsToNC3/HWToNC3
//     McToIo/STD <-> InputsFromNC3/NC3ToHW
//   XPlanar MC Project/Axes/Mover4330_1 <-> TcCOM Objects/XPlanar/Mover4330_1
//     IoToMc/STD <-> OutputsToNC3/HWToNC3
//     McToIo/STD <-> InputsFromNC3/NC3ToHW
//   XPlanar MC Project/Axes/Mover4550_1 <-> TcCOM Objects/XPlanar/Mover4550_1
//     IoToMc/STD <-> OutputsToNC3/HWToNC3
//     McToIo/STD <-> InputsFromNC3/NC3ToHW
//   PLC1/PLC1 Instance <-> XPlanar MC Project/Axes/Mover4220_1
//     PlcTask Inputs/MAIN.XPlanarModule.Mover[2]._Mover.MCTOPLC/ACT <-> McToPlc/ACT
//     PlcTask Inputs/MAIN.XPlanarModule.Mover[2]._Mover.MCTOPLC/COORDMODE <-> McToPlc/COORDMODE
//     PlcTask Inputs/MAIN.XPlanarModule.Mover[2]._Mover.MCTOPLC/SET <-> McToPlc/SET
//     PlcTask Inputs/MAIN.XPlanarModule.Mover[2]._Mover.MCTOPLC/SETONTRACK <-> McToPlc/SETONTRACK
//     PlcTask Inputs/MAIN.XPlanarModule.Mover[2]._Mover.MCTOPLC/STD <-> McToPlc/STD
//     PlcTask Outputs/MAIN.XPlanarModule.Mover[2]._Mover.PLCTOMC/STD <-> PlcToMc/STD
//   PLC1/PLC1 Instance <-> XPlanar MC Project/Axes/Mover4330_1
//     PlcTask Inputs/MAIN.XPlanarModule.Mover[1]._Mover.MCTOPLC/ACT <-> McToPlc/ACT
//     PlcTask Inputs/MAIN.XPlanarModule.Mover[1]._Mover.MCTOPLC/COORDMODE <-> McToPlc/COORDMODE
//     PlcTask Inputs/MAIN.XPlanarModule.Mover[1]._Mover.MCTOPLC/SET <-> McToPlc/SET
//     PlcTask Inputs/MAIN.XPlanarModule.Mover[1]._Mover.MCTOPLC/SETONTRACK <-> McToPlc/SETONTRACK
//     PlcTask Inputs/MAIN.XPlanarModule.Mover[1]._Mover.MCTOPLC/STD <-> McToPlc/STD
//     PlcTask Outputs/MAIN.XPlanarModule.Mover[1]._Mover.PLCTOMC/STD <-> PlcToMc/STD
//   PLC1/PLC1 Instance <-> XPlanar MC Project/Axes/Mover4550_1
//     PlcTask Inputs/MAIN.XPlanarModule.Mover[3]._Mover.MCTOPLC/ACT <-> McToPlc/ACT
//     PlcTask Inputs/MAIN.XPlanarModule.Mover[3]._Mover.MCTOPLC/COORDMODE <-> McToPlc/COORDMODE
//     PlcTask Inputs/MAIN.XPlanarModule.Mover[3]._Mover.MCTOPLC/SET <-> McToPlc/SET
//     PlcTask Inputs/MAIN.XPlanarModule.Mover[3]._Mover.MCTOPLC/SETONTRACK <-> McToPlc/SETONTRACK
//     PlcTask Inputs/MAIN.XPlanarModule.Mover[3]._Mover.MCTOPLC/STD <-> McToPlc/STD
//     PlcTask Outputs/MAIN.XPlanarModule.Mover[3]._Mover.PLCTOMC/STD <-> PlcToMc/STD
//   PLC1/PLC1 Instance <-> XPlanar MC Project/Groups/Environment
//     PlcTask Inputs/XPlanar.Environment.MCTOPLC_STD <-> McToPlc/STD
//   PLC1/PLC1 Instance <-> XPlanar MC Project/Groups/Track1
//     PlcTask Inputs/MAIN.XPlanarModule.Track[1]._Track.MCTOPLC_STD <-> McToPlc/STD
//   PLC1/PLC1 Instance <-> XPlanar MC Project/Groups/XPlanar
//     PlcTask Inputs/XPlanar.Group.MCTOPLC_STD <-> McToPlc/STD

CONFIGURATION PLC1
    RESOURCE PLC ON TwinCAT3
        TASK PlcTask(INTERVAL := T#10ms, PRIORITY := 20);
        PROGRAM MAIN WITH PlcTask : MAIN;
    END_RESOURCE
END_CONFIGURATION

// ---- POUs/MAIN.TcPOU
PROGRAM MAIN
VAR
	//Main machine module declaration
	XPlanarModule : FB_XPlanarModule;

	//Control Source for running machine
	ControlSourceHMI : FB_ControlSource;
	ControlSourcePB	 : FB_ControlSource;

	//Local Vars
	InitComplete : BOOL;
	_DCLinkOK	: BOOL;

END_VAR

CyclicLogic();

// Cope Resetting Code
IF XPlanarModule.InitComplete THEN
	
	CASE XPlanarModule.CurrentState OF
		
		// Aborting - wait for rising edge of DCLinkOK
		ePMLState_aborted:

			IF XPlanarModule.DC_Bus_OK AND NOT _DCLinkOK THEN
				XPlanarModule.ChangeState(ePMLCommand_Clear);
			END_IF

		ePMLState_Stopped:
			XPlanarModule.ChangeState(ePMLCommand_Reset);

		ePMLState_Idle:
			IF XPlanarModule._CommandedState = ePMLCommand_Clear THEN
				XPlanarModule.ChangeState(ePMLCommand_Reset);
			ELSIF XPlanarModule._CommandedState = ePMLCommand_Reset THEN
				XPlanarModule.ChangeState(ePMLCommand_Start);
			END_IF
	
	END_CASE

	// Save Previous Values
	_DCLinkOK	:= XPlanarModule.DC_Bus_OK;
END_IF

METHOD CyclicLogic
VAR_INPUT
END_VAR
IF NOT InitComplete THEN
	InitComplete := Initialize();
	RETURN;
END_IF

//Machine support HMI & Production Monitor
ControlSourcePB.CyclicLogic();
ControlSourceHMI.CyclicLogic();

//Machine Cyclic Logic
XPlanarModule.CyclicLogic();
END_METHOD

METHOD Initialize : BOOL
//Top level machine initialization should happen here, in the main initialization METHOD. Each subsequent "layer" OF modules will be named within their respective "parent" intialize METHOD
IF NOT ControlSourceHMI.Registered THEN
	XPlanarModule.RegisterExternalController(ControlSourceHMI);
END_IF

IF NOT ControlSourcePB.Registered THEN
	XPlanarModule.RegisterExternalController(ControlSourcePB);
END_IF

ControlSourceHMI.CyclicLogic();
ControlSourcePB.CyclicLogic();

//ADSLOGSTR(ADSLOG_MSGTYPE_WARN, 'Lag Monitoring disabled', 'For simulation demo only',);
Initialize := TRUE;
END_METHOD

END_PROGRAM

// ---- POUs/FB_XPlanarModule.TcPOU
FUNCTION_BLOCK FB_XPlanarModule EXTENDS FB_PackML_BaseModule
VAR
	// Component definitions here
	XPlanarTable : FB_Component_Xplanar := (Name := 'XPlanarTable');

	//Station Components
	Station1 : FB_RotateStation := (Name := 'Station1'); //Declaration of a custom station
	Station2 : FB_TiltStation 	:= (Name := 'Station2');
	Station3 : FB_BounceStation := (Name := 'Station3');

	//Helper Vars
	Mover			  : ARRAY[1..SystemParameters.MOVER_COUNT] OF FB_XPlanarMover;
	Track			  : ARRAY[1..SystemParameters.TRACK_COUNT] OF FB_XPlanarTrackSegment;
	TracksInitialized : BOOL;
END_VAR

VAR_OUTPUT
	DC_Bus_OK		: BOOL;
END_VAR

//! @summary This method contains code which will execute when this PackML module is in the <b>Aborting</b> state
METHOD PROTECTED Aborting
VAR
	i				: UDINT;
	SubModulesReady : BOOL := TRUE;
END_VAR
CASE DescendantSequenceState OF
	0:
		NoStateTasksToComplete := FALSE;
		NextStep(DescendantSequenceState);

	10:
		IF XPlanarTable.Abort() THEN
			StateTasksComplete := TRUE;
			NextStep(DescendantSequenceState);
		END_IF

	20:
		StateTasksComplete := TRUE;
END_CASE

SUPER^.Aborting();
END_METHOD

//! @summary This method contains code which will execute when this PackML module is in the <b>Clearing</b> state
METHOD PROTECTED Clearing
VAR
	i				: UDINT;
	SubModulesReady : BOOL := TRUE;
END_VAR

VAR_INST
	ipResult : I_PlanarTaskResult;
END_VAR

(*! <description> <b>Note:</b> The <i>Clear</i> command can also be thought of as a <i>fault reset</i> depite the ambiguity in the naming of the <i>Reset</i> state. 
<table> 
	<tr>
		<th> Previous State </th>
		<th> Transition In </th>
		<th> Transition Out </th>
		<th> Next State  </th> 
	</tr>
	<tr>
		<td> Aborted </td>
		<td> Clear Command </td> 
		<td> State Complete </td>
		<td> Stopped </td> 
	</tr>
</table>
This method is called as required by <c>StateControl()</c>
</description> 

*)
CASE _CurrentMode OF
	E_PMLUnitMode.ePMLUnitMode_Production:
		CASE DescendantSequenceState OF
			0: //Init
				NoStateTasksToComplete := FALSE;

				//Reset Stations
				Station1.Reset();
				Station2.Reset();
				Station3.Reset();
				NextStep(DescendantSequenceState);

			10: //Reset XPlanar System
				IF XPlanarTable.Reset() THEN
					NextStep(DescendantSequenceState);
				END_IF

			20: //Enable Group
				ipResult := XPlanarTable.EnableGroup();
				IF ipResult.Done THEN
					NextStep(DescendantSequenceState);
				ELSIF ipResult.Error THEN
					ErrorStep(DescendantSequenceState);
				END_IF

			30: //Clearing complete			
				StateTasksComplete := TRUE;
		END_CASE

	E_PMLUnitMode.ePMLUnitMode_Manual:
		;
END_CASE

SUPER^.Clearing();
END_METHOD

METHOD CyclicLogic
VAR
	i : INT;
END_VAR
IF NOT _InitComplete THEN
	_InitComplete := Initialize();
END_IF

//Add any required cyclic logic here

//Call the base logic
SUPER^.CyclicLogic();


DC_Bus_OK	:= XPlanar.Tiles[1].DcLinkOk;
END_METHOD

//! @summary This method contains code which will execute when this PackML module is in the <b>Execute</b> state
METHOD PROTECTED Execute
VAR
	i : UDINT;
END_VAR
CASE _CurrentMode OF
	E_PMLUnitMode.ePMLUnitMode_Production:
		FOR i := 1 TO SystemParameters.STATION_COUNT DO
			ip.Stations[i].Execute();
		END_FOR

	E_PMLUnitMode.ePMLUnitMode_Manual:
		; //Insert logic for Manual Mode here
END_CASE
END_METHOD

//! @summary Automatically enables and disables HMI control based on the PackML mode
METHOD PROTECTED HMIPermissions

//! @description This method is called cyclically by <c>CyclicLogic()</c>
//General Mode Based Monitoring and handling of HMI control
CASE _CurrentMode OF
	E_PMLUnitMode.ePMLUnitMode_Production:
		AllowHMIControl(ThisModuleOnly := FALSE);

	E_PMLUnitMode.ePMLUnitMode_Manual:
		AllowHMIControl(ThisModuleOnly := FALSE);

	E_PMLUnitMode.ePMLUnitMode_Maintenance:
		AllowHMIControl(ThisModuleOnly := FALSE);
END_CASE
END_METHOD

//! @summary Basic module initialization logic
METHOD PROTECTED Initialize : BOOL;
VAR
	i						 : UDINT;
	varInfo					 : __SYSTEM.VAR_INFO;
	AllSubUnitsInitialized	 : BOOL := TRUE;
	AllComponentsInitialized : BOOL := TRUE;
END_VAR

//! @description This method is called by <c>CyclicLogic()</c> as required
Initialize := FALSE;
CASE DescendantSequenceState OF
	0: //Register Submodules and Components
		RegisterComponent(XPlanarTable);
		RegisterComponent(Station1);
		RegisterComponent(Station2);
		RegisterComponent(Station3);
		_LogModeChanges			:= FALSE;
		_LogStateChanges		:= FALSE;
		DescendantSequenceState := DescendantSequenceState + 10;

	10: //Set interfaces *This must be done before initializing the base class!

		//Set mover interfaces
		FOR i := 1 TO SystemParameters.MOVER_COUNT DO
			Mover[i].MoverIndex := i;
			ip.Movers[i]		:= Mover[i];
		END_FOR

		//Set Track Interfaces
		FOR i := 1 TO SystemParameters.TRACK_COUNT DO
			ip.Tracks[i] := Track[i];
		END_FOR

		//Set Station interfaces
		ip.Stations[1]			:= Station1;
		ip.Stations[2]			:= Station2;
		ip.Stations[3]			:= Station3;
		DescendantSequenceState := DescendantSequenceState + 10;

	20: //Call Initialize of the base class
		IF SUPER^.Initialize() THEN
			DescendantSequenceState := DescendantSequenceState + 10;
		END_IF

	30:
		Initialize := TRUE;
END_CASE
END_METHOD

METHOD PROTECTED Resetting
VAR_INST
	i			 : UDINT;
	ipTaskResult : I_PlanarTaskResult;
END_VAR
CASE _CurrentMode OF
	E_PMLUnitMode.ePMLUnitMode_Production:
		CASE DescendantSequenceState OF
			0: //Init
				i					   := 1;
				NoStateTasksToComplete := FALSE;
				NextStep(DescendantSequenceState);

			10: //Enable Tracks
				ipTaskResult := XplanarTable.EnableTracks();
				IF ipTaskResult.Done THEN
					NextStep(DescendantSequenceState);
				ELSIF ipTaskResult.Error THEN //An error occured, jump to 'error step'
					ErrorStep(DescendantSequenceState);
				END_IF

			20: //Enable Movers
				ipTaskResult := XPlanarTable.EnableMovers();
				IF ipTaskResult.Done THEN
					NextStep(DescendantSequenceState);
				ELSIF ipTaskResult.Error THEN //An error occured, jump to 'error step'
					ErrorStep(DescendantSequenceState);
				END_IF

			30: //Add Tracks to Group
				ipTaskResult := XPlanarTable.AddTracksToGroup();
				IF ipTaskResult.Done THEN
					NextStep(DescendantSequenceState);
				ELSIF ipTaskResult.Error THEN //An error occured, jump to 'error step'
					ErrorStep(DescendantSequenceState);
				END_IF

			40: //Add Movers to Group			
				ipTaskResult := XPlanarTable.AddMoversToGroup();
				IF ipTaskResult.Done THEN
					NextStep(DescendantSequenceState);
				ELSIF ipTaskResult.Error THEN //An error occured, jump to 'error step'
					ErrorStep(DescendantSequenceState);
				END_IF

			50: //Clearing complete
				StateTasksComplete := TRUE;
		END_CASE
END_CASE

SUPER^.Resetting();
END_METHOD

METHOD PRIVATE SetupStations : BOOL
VAR_INPUT
END_VAR
//Set Required Process Station Initialization Parameters
Station1.Position.SetValuesXYC(240, 120, 0);
Station1.Size.x		   := 120;		//Changes the station size in the X plane (optional - Default is 120mm)
Station1.Size.y		   := 120;		//Changes the station size in the Y plane (optionsl- Default is 120mm)
Station1.TrackID	   := 1;		//Set Index of the track segment the station resides on if applicable	
Station1.NextStation   := Station2; //Set the interface for the next station of the mover
Station1.StationAngle  := 180;
Station1.NumberOfTurns := 2;

Station2.Position.SetValuesXYC(240, 600, 0);
Station2.TrackID	   := 1;
Station2.NextStation   := Station3;
Station2.StationAngle  := 3.0;

Station3.Position.SetValuesXYC(360, 360, 0);
Station3.TrackID	   := 1;
Station3.NextStation   := Station1;
Station3.StationAngle  := -90;

//Return TRUE when all necessary station parameters are set
SetupStations := TRUE;
END_METHOD

METHOD PROTECTED Starting
VAR_INST
	i		  : UDINT;
	ipResult  : I_PlanarTaskResult;
	InitTimer : TON;
END_VAR
CASE _CurrentMode OF
	E_PMLUnitMode.ePMLUnitMode_Production:
		CASE DescendantSequenceState OF
			0:
				NoStateTasksToComplete	:= FALSE;
				DescendantSequenceState := 10;
				i						:= 1;

			10: //Set Station Parameters
				SetupStations();
				NextStep(DescendantSequenceState);

			20: //Cleanup mover queues
				FOR i := 1 TO SystemParameters.STATION_COUNT DO
					ip.Stations[i].MoverQueue.Dequeue();
				END_FOR

				NextStep(DescendantSequenceState);

			30: //Set some initial application move dynamics
				FOR i := 1 TO SystemParameters.MOVER_COUNT DO
					ip.Movers[i].Dynamics.Movement.Accel	:= 2000;
					ip.Movers[i].Dynamics.Movement.Decel	:= 2000;
					ip.Movers[i].Dynamics.Movement.Velocity := 300;
					ip.Movers[i].Dynamics.Movement.Jerk		:= 50000;
					ip.Movers[i].Dynamics.Rotation.Accel	:= 5000;
					ip.Movers[i].Dynamics.Rotation.Decel	:= 5000;
					ip.Movers[i].Dynamics.Rotation.Velocity := 300;
					ip.Movers[i].Dynamics.Rotation.Jerk		:= 100000;
					ip.Movers[i].Dynamics.Tilt.Accel		:= 5000;
					ip.Movers[i].Dynamics.Tilt.Decel		:= 5000;
					ip.Movers[i].Dynamics.Tilt.Velocity		:= 300;
					ip.Movers[i].Dynamics.Tilt.Jerk			:= 100000;
					ip.Movers[i].Gap						:= 400;
					ip.Movers[i].Destination				:= 0;
				END_FOR

				i := 1;
				NextStep(DescendantSequenceState);

			40: //Square Up movers
				IF i <= SystemParameters.MOVER_COUNT THEN
					ipResult := ip.Movers[i].MoveCommand.SquareUp();
					IF ipResult.Done THEN
						NextMinorStep(DescendantSequenceState);
					ELSIF ipResult.Error THEN
						ErrorStep(DescendantSequenceState);
					END_IF
				ELSE
					i := 1;
					NextStep(DescendantSequenceState);
				END_IF				

			41: //Check Mover Count
				IF i <= SystemParameters.MOVER_COUNT THEN
					i						:= i + 1;
					DescendantSequenceState := 40;
				ELSE
					i := 1;
					NextStep(DescendantSequenceState);
				END_IF

			50: //Join Movers to nearest track
				IF i <= SystemParameters.MOVER_COUNT THEN
					ipResult := ip.Movers[i].MoveCommand.JoinClosestTrack(FALSE);
					IF ipResult.Done THEN
						NextMinorStep(DescendantSequenceState);
					ELSIF ipResult.Error THEN
						ErrorStep(DescendantSequenceState);
					END_IF
				ELSE
					i := 1;
					NextStep(DescendantSequenceState);
				END_IF

			51: //Check Mover Count
				IF i <= SystemParameters.MOVER_COUNT THEN
					i						:= i + 1;
					DescendantSequenceState := 50;
				ELSE
					i := 1;
					NextStep(DescendantSequenceState);
				END_IF

			60: //Send Movers around to station 1
				IF i <= SystemParameters.MOVER_COUNT THEN
					ipResult := ip.Movers[i].MoveCommand.SendToStation(ip.Stations[1]);
					IF ipResult.Busy THEN
						NextMinorStep(DescendantSequenceState);
					ELSIF ipResult.Error THEN
						ErrorStep(DescendantSequenceState);
					END_IF
				ELSE
					i := 1;
					NextStep(DescendantSequenceState);
				END_IF

			61: //Check Mover Count
				IF i <= SystemParameters.MOVER_COUNT THEN
					i						:= i + 1;
					DescendantSequenceState := 60;
				ELSE
					i := 1;
					NextStep(DescendantSequenceState);
				END_IF

			70: //Let recovery get moving before jumping to execute
				InitTimer(IN := TRUE, PT := T#500MS);
				IF InitTimer.Q THEN
					InitTimer(IN := FALSE);
					StateTasksComplete := TRUE;
				END_IF
		END_CASE

	E_PMLUnitMode.ePMLUnitMode_Manual:
		;
END_CASE

SUPER^.Starting();
END_METHOD

END_FUNCTION_BLOCK

// ---- POUs/CustomStations/FB_TiltStation.TcPOU
FUNCTION_BLOCK FB_TiltStation EXTENDS FB_XPlanarStationBase
VAR
	_StationAngle  : LREAL;
	ProcessState	: INT;
	ProcessStateOld	: INT;
	TON_StateChange	: TON := (PT := T#100MS);
	CommandResultDone	: BOOL;
	TiltAngle		: LREAL;
END_VAR

METHOD Execute
VAR_INST
	i			  : UDINT := 1;
	CommandResult : I_PlanarTaskResult;
END_VAR
SUPER^.Execute();
IF StationState = E_XPlanarStationState.ProcessMover THEN
	CASE ProcessState OF

		0:	// Raise Z
			CommandResult		:= ipCurrentMover.MoveCommand.VerticalMove(5.0);
			IF ipCurrentMover.MoverType = APM4220 THEN
				TiltAngle		:= 4.5;
			ELSIF ipCurrentMOVER.MoverType = APM4330 THEN
				TiltAngle		:= 3.0;
			ELSIF ipCurrentMover.MoverType = APM4550 THEN
				TiltAngle		:= 2.0;
			END_IF
			ProcessState		:= 1;

		1:	// Check for Result
			IF CommandResult.Done AND TON_StateChange.Q THEN
				ProcessState 	:= 2;
			END_IF

		2:	// Tilt A Positive
			CommandResult		:= ipCurrentMover.MoveCommand.TiltA(TiltAngle);
			ProcessState 		:= 3;

		3:	// Check for Result
			IF CommandResult.Done AND TON_StateChange.Q THEN
				ProcessState	:= 4;
			END_IF
			
		4:	// Tilt A Negative
			CommandResult		:= ipCurrentMover.MoveCommand.TiltA(TiltAngle * -1.0);
			ProcessState 		:= 5;

		5:	// Check for Result
			IF CommandResult.Done AND TON_StateChange.Q THEN
				ProcessState	:= 6;
			END_IF
			
		6:	// Tilt A Zero
			CommandResult		:= ipCurrentMover.MoveCommand.TiltA(0.0);
			ProcessState		:= 7;

		7:	// Check for Result
			IF CommandResult.Done AND TON_StateChange.Q THEN
				ProcessState	:= 8;
			END_IF
			
		8:	// Tilt B Positive
			CommandResult		:= ipCurrentMover.MoveCommand.TiltB(TiltAngle);
			ProcessState 		:= 9;

		9:	// Check for Result
			IF CommandResult.Done AND TON_StateChange.Q THEN
				ProcessState	:= 10;
			END_IF
			
		10:	// Tilt B Negative
			CommandResult		:= ipCurrentMover.MoveCommand.TiltB(TiltAngle * -1.0);
			ProcessState 		:= 11;

		11:	// Check for Result
			IF CommandResult.Done AND TON_StateChange.Q THEN
				ProcessState 	:= 12;
			END_IF
			
		12:	// Tilt B Zero
			CommandResult		:= ipCurrentMover.MoveCommand.TiltB(0.0);
			ProcessState 		:= 13;

		13:	// Check for Result
			IF CommandResult.Done AND TON_StateChange.Q THEN
				ProcessState 	:= 14;
			END_IF

		14:	// Lower Z
			CommandResult		:= ipCurrentMover.MoveCommand.VerticalMove(2.0);
			ProcessState 		:= 15;

		15:	// Check for Result
			IF CommandResult.Done AND TON_StateChange.Q THEN
				ProcessState 	:= 16;
			END_IF

		16:	// Done
			_StationComplete 	:= TRUE;

	END_CASE

	// Timer Call
	TON_StateChange(IN := ProcessState = ProcessStateOld);

ELSE
	ProcessState	:= 0;
	TON_StateChange(IN := FALSE);

END_IF

// Save Prevoius Values
ProcessStateOld	:= ProcessState;

// Debug
IF CommandResult <> 0 THEN
	CommandResultDone	:= CommandResult.Done;
ELSE
	CommandResultDone	:= FALSE;
END_IF
END_METHOD

PROPERTY StationAngle : LREAL
SET
_StationAngle := StationAngle;
END_SET
END_PROPERTY

END_FUNCTION_BLOCK

// ---- POUs/CustomStations/FB_BounceStation.TcPOU
FUNCTION_BLOCK FB_BounceStation EXTENDS FB_XPlanarStationBase
VAR
	_StationAngle  : LREAL;
	ProcessState	: INT;
	ProcessStateOld	: INT;
	TON_StateChange	: TON := (PT := T#100MS);
	CommandResultDone	: BOOL;
END_VAR

METHOD Execute
VAR_INST
	i			  : UDINT := 1;
	CommandResult : I_PlanarTaskResult;
END_VAR
SUPER^.Execute();
IF StationState = E_XPlanarStationState.ProcessMover THEN
	CASE ProcessState OF

		0:	// Move Z
			CommandResult		:= ipCurrentMover.MoveCommand.VerticalMove(3.0);
			ProcessState		:= 1;

		1:	// Check for Result
			IF CommandResult.Done AND TON_StateChange.Q THEN
				ProcessState 	:= 2;
			END_IF

		2:	// Move Z
			CommandResult		:= ipCurrentMover.MoveCommand.VerticalMove(1.0);
			ProcessState 		:= 3;

		3:	// Check for Result
			IF CommandResult.Done AND TON_StateChange.Q THEN
				ProcessState	:= 4;
			END_IF
			
		4:	// Move Z
			CommandResult		:= ipCurrentMover.MoveCommand.VerticalMove(4.0);
			ProcessState 		:= 5;

		5:	// Check for Result
			IF CommandResult.Done AND TON_StateChange.Q THEN
				ProcessState	:= 6;
			END_IF
			
		6:	// Move Z
			CommandResult		:= ipCurrentMover.MoveCommand.VerticalMove(1.0);
			ProcessState		:= 7;

		7:	// Check for Result
			IF CommandResult.Done AND TON_StateChange.Q THEN
				ProcessState	:= 8;
			END_IF
			
		8:	// Move Z
			CommandResult		:= ipCurrentMover.MoveCommand.VerticalMove(5.0);
			ProcessState 		:= 9;

		9:	// Check for Result
			IF CommandResult.Done AND TON_StateChange.Q THEN
				ProcessState	:= 10;
			END_IF
			
		10:	// Move Z
			CommandResult		:= ipCurrentMover.MoveCommand.VerticalMove(1.0);
			ProcessState 		:= 11;

		11:	// Check for Result
			IF CommandResult.Done AND TON_StateChange.Q THEN
				ProcessState 	:= 12;
			END_IF
			
		12:	// Move Z
			CommandResult		:= ipCurrentMover.MoveCommand.VerticalMove(6.0);
			ProcessState 		:= 13;

		13:	// Check for Result
			IF CommandResult.Done AND TON_StateChange.Q THEN
				ProcessState 	:= 14;
			END_IF

		14:	// Move Z
			CommandResult		:= ipCurrentMover.MoveCommand.VerticalMove(2.0);
			ProcessState 		:= 15;

		15:	// Check for Result
			IF CommandResult.Done AND TON_StateChange.Q THEN
				ProcessState 	:= 16;
			END_IF

		16:	// Done
			_StationComplete 	:= TRUE;

	END_CASE

	// Timer Call
	TON_StateChange(IN := ProcessState = ProcessStateOld);

ELSE
	ProcessState	:= 0;
	TON_StateChange(IN := FALSE);

END_IF

// Save Prevoius Values
ProcessStateOld	:= ProcessState;

// Debug
IF CommandResult <> 0 THEN
	CommandResultDone	:= CommandResult.Done;
ELSE
	CommandResultDone	:= FALSE;
END_IF
END_METHOD

PROPERTY StationAngle : LREAL
SET
_StationAngle := StationAngle;
END_SET
END_PROPERTY

END_FUNCTION_BLOCK

// ---- VISUs/V_Main.TcVIS
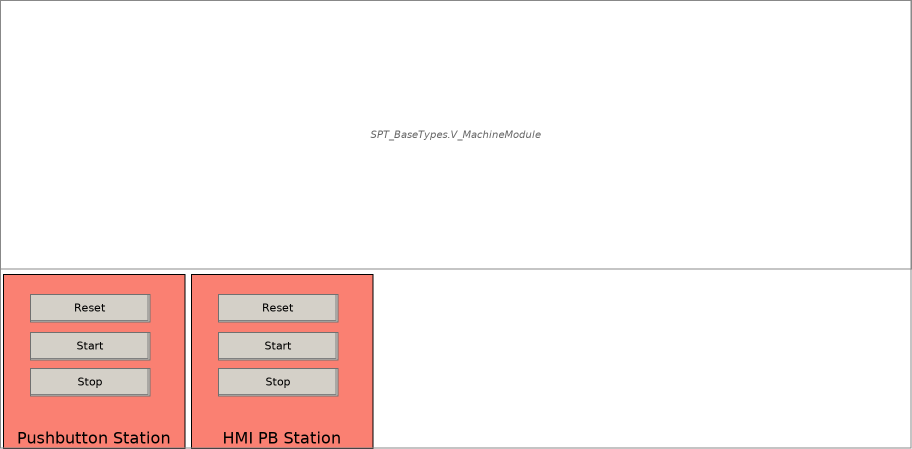
VISUALIZATION V_Main  // 912x449
    Frame (0,0 912x269)
        shows SPT_BaseTypes.V_MachineModule(HMI := MAIN.XPlanarModule.PackMLBaseModule_HMI)
    Group (3,274 182x175)
        RoundedRectangle (0,0 182x175), "Pushbutton Station"
        Button (27,94 120x28), "Stop", input disabled if: not MAIN.ControlSourcePB.MainPMLControl_Simplified.StopPermissive
            tap MAIN.ControlSourcePB.MainPMLControl_Simplified.StopPressed
        Button (27,20 120x28), "Reset", input disabled if: not MAIN.ControlSourcePB.MainPMLControl_Simplified.ResetPermissive
            tap MAIN.ControlSourcePB.MainPMLControl_Simplified.ResetPressed
        Button (27,58 120x28), "Start", input disabled if: not MAIN.ControlSourcePB.MainPMLControl_Simplified.StartPermissive
            tap MAIN.ControlSourcePB.MainPMLControl_Simplified.StartPressed
    Group (191,274 182x175)
        RoundedRectangle (0,0 182x175), "HMI PB Station"
        Button (27,94 120x28), "Stop", input disabled if: not MAIN.ControlSourceHMI.MainPMLControl_Simplified.StopPermissive
            tap MAIN.ControlSourceHMI.MainPMLControl_Simplified.StopPressed
        Button (27,20 120x28), "Reset", input disabled if: not MAIN.ControlSourceHMI.MainPMLControl_Simplified.ResetPermissive
            tap MAIN.ControlSourceHMI.MainPMLControl_Simplified.ResetPressed
        Button (27,58 120x28), "Start", input disabled if: not MAIN.ControlSourceHMI.MainPMLControl_Simplified.StartPermissive
            tap MAIN.ControlSourceHMI.MainPMLControl_Simplified.StartPressed
END_VISUALIZATION
